LIN {X 0,Y 328.019,Z 1054.025,A -85,B 0,C 180,E1 16291.397,E2 16291.397} C_VEL
LIN {X 0,Y 327.98,Z 1054.756,A -85,B 0,C 180,E1 16287.554,E2 16287.554} C_VEL
LIN {X 0,Y 328.061,Z 1053.985,A -85,B 0,C 180,E1 16283.525,E2 16283.525} C_VEL
LIN {X 0,Y 328.284,Z 1052.234,A -85,B 0,C 180,E1 16280.002,E2 16280.002} C_VEL
LIN {X 0,Y 329.029,Z 1048.812,A -85,B 0,C 180,E1 16275.794,E2 16275.794} C_VEL
LIN {X 0,Y 330.509,Z 1043.751,A -85,B 0,C 180,E1 16271.661,E2 16271.661} C_VEL
LIN {X 0,Y 332.865,Z 1037.506,A -85,B 0,C 180,E1 16267.699,E2 16267.699} C_VEL
LIN {X 0,Y 336.502,Z 1029.05,A -85,B 0,C 180,E1 16263.531,E2 16263.531} C_VEL
LIN {X 0,Y 340.822,Z 1020.018,A -85,B 0,C 180,E1 16259.889,E2 16259.889} C_VEL
LIN {X 0,Y 346.797,Z 1008.189,A -85,B 0,C 180,E1 16255.99,E2 16255.99} C_VEL
LIN {X 0,Y 352.877,Z 996.469,A -85,B 0,C 180,E1 16252.772,E2 16252.772} C_VEL
LIN {X 0,Y 360.668,Z 981.476,A -85,B 0,C 180,E1 16249.345,E2 16249.345} C_VEL
LIN {X 0,Y 367.6,Z 967.844,A -85,B 0,C 180,E1 16246.729,E2 16246.729} C_VEL
LIN {X 0,Y 376.145,Z 950.498,A -85,B 0,C 180,E1 16243.914,E2 16243.914} C_VEL
LIN {X 0,Y 383.701,Z 934.237,A -85,B 0,C 180,E1 16241.704,E2 16241.704} C_VEL
LIN {X 0,Y 392.054,Z 915.275,A -85,B 0,C 180,E1 16239.512,E2 16239.512} C_VEL
LIN {X 0,Y 397.893,Z 900.897,A -85,B 0,C 180,E1 16238.1,E2 16238.1} C_VEL
LIN {X 0,Y 399.57,Z 894.838,A -85,B 0,C 180,E1 16237.443,E2 16237.443} C_VEL
LIN {X 0,Y 401.539,Z 880.043,A -85,B 0,C 180,E1 16235.512,E2 16235.512} C_VEL
LIN {X 0,Y 403.175,Z 873.668,A -85,B 0,C 180,E1 16234.932,E2 16234.932} C_VEL
LIN {X 0,Y 409.897,Z 853.186,A -85,B 0,C 180,E1 16233.587,E2 16233.587} C_VEL
LIN {X 0,Y 416.193,Z 831.541,A -85,B 0,C 180,E1 16232.395,E2 16232.395} C_VEL
LIN {X 0,Y 421.864,Z 808.1,A -85,B 0,C 180,E1 16231.367,E2 16231.367} C_VEL
LIN {X 0,Y 426.386,Z 785.736,A -85,B 0,C 180,E1 16230.586,E2 16230.586} C_VEL
LIN {X 0,Y 430.208,Z 760.734,A -85,B 0,C 180,E1 16229.93,E2 16229.93} C_VEL
LIN {X 0,Y 432.597,Z 738.268,A -85,B 0,C 180,E1 16229.491,E2 16229.491} C_VEL
LIN {X 0,Y 447.979,Z 526.259,A -85,B 0,C 180,E1 16226.067,E2 16226.067} C_VEL
LIN {X 0,Y 439.532,Z 512.486,A -85,B 0,C 180,E1 16223.283,E2 16223.283} C_VEL
LIN {X 0,Y 431.504,Z 500.147,A -85,B 0,C 180,E1 16220.234,E2 16220.234} C_VEL
LIN {X 0,Y 424.951,Z 490.677,A -85,B 0,C 180,E1 16217.317,E2 16217.317} C_VEL
LIN {X 0,Y 420.889,Z 485.14,A -85,B 0,C 180,E1 16215.219,E2 16215.219} C_VEL
LIN {X 0,Y 417.649,Z 480.579,A -85,B 0,C 180,E1 16213.287,E2 16213.287} C_VEL
LIN {X 0,Y 414.017,Z 475.592,A -85,B 0,C 180,E1 16210.717,E2 16210.717} C_VEL
LIN {X 0,Y 410.905,Z 471.414,A -85,B 0,C 180,E1 16207.902,E2 16207.902} C_VEL
LIN {X 0,Y 410.246,Z 470.248,A -85,B 0,C 180,E1 16207.141,E2 16207.141} C_VEL
LIN {X 0,Y 406.911,Z 465.074,A -85,B 0,C 180,E1 16199.437,E2 16199.437} C_VEL
LIN {X 0,Y 406.969,Z 465.799,A -85,B 0,C 180,E1 16197.606,E2 16197.606} C_VEL
LIN {X 0,Y 410.641,Z 470.746,A -85,B 0,C 180,E1 16190.752,E2 16190.752} C_VEL
LIN {X 0,Y 413.009,Z 474.635,A -85,B 0,C 180,E1 16188.408,E2 16188.408} C_VEL
LIN {X 0,Y 414.68,Z 476.395,A -85,B 0,C 180,E1 16187.112,E2 16187.112} C_VEL
LIN {X 0,Y 418.024,Z 480.996,A -85,B 0,C 180,E1 16184.816,E2 16184.816} C_VEL
LIN {X 0,Y 422.672,Z 487.53,A -85,B 0,C 180,E1 16182.16,E2 16182.16} C_VEL
LIN {X 0,Y 426.717,Z 493.371,A -85,B 0,C 180,E1 16180.173,E2 16180.173} C_VEL
LIN {X 0,Y 433.716,Z 505.116,A -85,B 0,C 180,E1 16177.141,E2 16177.141} C_VEL
LIN {X 0,Y 441.286,Z 518.517,A -85,B 0,C 180,E1 16174.32,E2 16174.32} C_VEL
LIN {X 0,Y 447.828,Z 531.14,A -85,B 0,C 180,E1 16172.136,E2 16172.136} C_VEL
LIN {X 0,Y 431.317,Z 757.329,A -85,B 0,C 180,E1 16168.476,E2 16168.476} C_VEL
LIN {X 0,Y 427.838,Z 784.421,A -85,B 0,C 180,E1 16167.9,E2 16167.9} C_VEL
LIN {X 0,Y 423.888,Z 806.262,A -85,B 0,C 180,E1 16167.286,E2 16167.286} C_VEL
LIN {X 0,Y 418.06,Z 831.955,A -85,B 0,C 180,E1 16166.338,E2 16166.338} C_VEL
LIN {X 0,Y 412.513,Z 852.441,A -85,B 0,C 180,E1 16165.378,E2 16165.378} C_VEL
LIN {X 0,Y 405.328,Z 875.569,A -85,B 0,C 180,E1 16164.047,E2 16164.047} C_VEL
LIN {X 0,Y 398.484,Z 894.862,A -85,B 0,C 180,E1 16162.696,E2 16162.696} C_VEL
LIN {X 0,Y 390.831,Z 914.648,A -85,B 0,C 180,E1 16161.055,E2 16161.055} C_VEL
LIN {X 0,Y 382.147,Z 934.931,A -85,B 0,C 180,E1 16159.013,E2 16159.013} C_VEL
LIN {X 0,Y 374.49,Z 951.703,A -85,B 0,C 180,E1 16157.019,E2 16157.019} C_VEL
LIN {X 0,Y 365.624,Z 969.96,A -85,B 0,C 180,E1 16154.435,E2 16154.435} C_VEL
LIN {X 0,Y 357.949,Z 985.105,A -85,B 0,C 180,E1 16151.884,E2 16151.884} C_VEL
LIN {X 0,Y 349.451,Z 1001.499,A -85,B 0,C 180,E1 16148.592,E2 16148.592} C_VEL
LIN {X 0,Y 342.714,Z 1014.35,A -85,B 0,C 180,E1 16145.492,E2 16145.492} C_VEL
LIN {X 0,Y 336.074,Z 1027.324,A -85,B 0,C 180,E1 16141.777,E2 16141.777} C_VEL
LIN {X 0,Y 330.792,Z 1038.04,A -85,B 0,C 180,E1 16138.038,E2 16138.038} C_VEL
LIN {X 0,Y 326.517,Z 1047.639,A -85,B 0,C 180,E1 16134.034,E2 16134.034} C_VEL
LIN {X 0,Y 323.393,Z 1055.523,A -85,B 0,C 180,E1 16129.883,E2 16129.883} C_VEL
LIN {X 0,Y 321.47,Z 1061.654,A -85,B 0,C 180,E1 16125.885,E2 16125.885} C_VEL
LIN {X 0,Y 320.346,Z 1066.696,A -85,B 0,C 180,E1 16121.453,E2 16121.453} C_VEL
LIN {X 0,Y 319.995,Z 1069.639,A -85,B 0,C 180,E1 16117.722,E2 16117.722} C_VEL
LIN {X 0,Y 319.957,Z 1071.386,A -85,B 0,C 180,E1 16114.122,E2 16114.122} C_VEL
LIN {X 0,Y 319.988,Z 1072.022,A -85,B 0,C 180,E1 16110.179,E2 16110.179} C_VEL
LIN {X 0,Y 319.968,Z 1071.269,A -85,B 0,C 180,E1 16106.417,E2 16106.417} C_VEL
LIN {X 0,Y 319.984,Z 1069.557,A -85,B 0,C 180,E1 16103,E2 16103} C_VEL
LIN {X 0,Y 320.217,Z 1066.668,A -85,B 0,C 180,E1 16099.384,E2 16099.384} C_VEL
LIN {X 0,Y 321.182,Z 1061.399,A -85,B 0,C 180,E1 16094.841,E2 16094.841} C_VEL
LIN {X 0,Y 322.786,Z 1055.481,A -85,B 0,C 180,E1 16091.019,E2 16091.019} C_VEL
LIN {X 0,Y 325.582,Z 1047.504,A -85,B 0,C 180,E1 16086.853,E2 16086.853} C_VEL
LIN {X 0,Y 329.389,Z 1038.022,A -85,B 0,C 180,E1 16082.913,E2 16082.913} C_VEL
LIN {X 0,Y 334.287,Z 1027.212,A -85,B 0,C 180,E1 16079.144,E2 16079.144} C_VEL
LIN {X 0,Y 340.353,Z 1014.354,A -85,B 0,C 180,E1 16075.459,E2 16075.459} C_VEL
LIN {X 0,Y 346.711,Z 1001.36,A -85,B 0,C 180,E1 16072.31,E2 16072.31} C_VEL
LIN {X 0,Y 354.366,Z 985.586,A -85,B 0,C 180,E1 16069.109,E2 16069.109} C_VEL
LIN {X 0,Y 361.656,Z 970.313,A -85,B 0,C 180,E1 16066.495,E2 16066.495} C_VEL
LIN {X 0,Y 370.629,Z 950.761,A -85,B 0,C 180,E1 16063.696,E2 16063.696} C_VEL
LIN {X 0,Y 377.757,Z 934.31,A -85,B 0,C 180,E1 16061.718,E2 16061.718} C_VEL
LIN {X 0,Y 386.147,Z 913.615,A -85,B 0,C 180,E1 16059.615,E2 16059.615} C_VEL
LIN {X 0,Y 392.979,Z 895.121,A -85,B 0,C 180,E1 16058.049,E2 16058.049} C_VEL
LIN {X 0,Y 400.135,Z 874.089,A -85,B 0,C 180,E1 16056.545,E2 16056.545} C_VEL
LIN {X 0,Y 406.584,Z 852.194,A -85,B 0,C 180,E1 16055.267,E2 16055.267} C_VEL
LIN {X 0,Y 411.987,Z 831.39,A -85,B 0,C 180,E1 16054.268,E2 16054.268} C_VEL
LIN {X 0,Y 417.472,Z 806.131,A -85,B 0,C 180,E1 16053.315,E2 16053.315} C_VEL
LIN {X 0,Y 421.276,Z 784.291,A -85,B 0,C 180,E1 16052.684,E2 16052.684} C_VEL
LIN {X 0,Y 424.587,Z 757.418,A -85,B 0,C 180,E1 16052.1,E2 16052.1} C_VEL
LIN {X 0,Y 440.37,Z 531.132,A -85,B 0,C 180,E1 16048.393,E2 16048.393} C_VEL
LIN {X 0,Y 440.634,Z 526.173,A -85,B 0,C 180,E1 16048.293,E2 16048.293} C_VEL
LIN {X 0,Y 432.575,Z 510.753,A -85,B 0,C 180,E1 16045.794,E2 16045.794} C_VEL
LIN {X 0,Y 424.816,Z 497.033,A -85,B 0,C 180,E1 16043.109,E2 16043.109} C_VEL
LIN {X 0,Y 418.086,Z 485.932,A -85,B 0,C 180,E1 16040.473,E2 16040.473} C_VEL
LIN {X 0,Y 412.337,Z 477.708,A -85,B 0,C 180,E1 16037.937,E2 16037.937} C_VEL
LIN {X 0,Y 407.928,Z 471.833,A -85,B 0,C 180,E1 16035.715,E2 16035.715} C_VEL
LIN {X 0,Y 404.622,Z 467.31,A -85,B 0,C 180,E1 16033.796,E2 16033.796} C_VEL
LIN {X 0,Y 401.321,Z 462.864,A -85,B 0,C 180,E1 16031.57,E2 16031.57} C_VEL
LIN {X 0,Y 397.458,Z 458.072,A -85,B 0,C 180,E1 16028.317,E2 16028.317} C_VEL
LIN {X 0,Y 396.63,Z 456.484,A -85,B 0,C 180,E1 16027.387,E2 16027.387} C_VEL
LIN {X 0,Y 393.119,Z 452.323,A -85,B 0,C 180,E1 16021.457,E2 16021.457} C_VEL
LIN {X 0,Y 392.894,Z 450.705,A -85,B 0,C 180,E1 16018.833,E2 16018.833} C_VEL
LIN {X 0,Y 393.131,Z 452.387,A -85,B 0,C 180,E1 16016.062,E2 16016.062} C_VEL
LIN {X 0,Y 396.418,Z 456.356,A -85,B 0,C 180,E1 16010.417,E2 16010.417} C_VEL
LIN {X 0,Y 397.008,Z 457.086,A -85,B 0,C 180,E1 16009.772,E2 16009.772} C_VEL
LIN {X 0,Y 399.817,Z 461.29,A -85,B 0,C 180,E1 16007.139,E2 16007.139} C_VEL
LIN {X 0,Y 401.324,Z 462.818,A -85,B 0,C 180,E1 16006.015,E2 16006.015} C_VEL
LIN {X 0,Y 404.74,Z 467.435,A -85,B 0,C 180,E1 16003.716,E2 16003.716} C_VEL
LIN {X 0,Y 409.748,Z 474.244,A -85,B 0,C 180,E1 16000.913,E2 16000.913} C_VEL
LIN {X 0,Y 413.929,Z 480.014,A -85,B 0,C 180,E1 15998.904,E2 15998.904} C_VEL
LIN {X 0,Y 419.585,Z 487.91,A -85,B 0,C 180,E1 15996.511,E2 15996.511} C_VEL
LIN {X 0,Y 428.149,Z 500.756,A -85,B 0,C 180,E1 15993.359,E2 15993.359} C_VEL
LIN {X 0,Y 436.584,Z 514.241,A -85,B 0,C 180,E1 15990.652,E2 15990.652} C_VEL
LIN {X 0,Y 440.881,Z 521.726,A -85,B 0,C 180,E1 15989.377,E2 15989.377} C_VEL
LIN {X 0,Y 425.191,Z 745.395,A -85,B 0,C 180,E1 15985.721,E2 15985.721} C_VEL
LIN {X 0,Y 421.987,Z 771.99,A -85,B 0,C 180,E1 15985.121,E2 15985.121} C_VEL
LIN {X 0,Y 418.53,Z 792.778,A -85,B 0,C 180,E1 15984.488,E2 15984.488} C_VEL
LIN {X 0,Y 413.739,Z 816.139,A -85,B 0,C 180,E1 15983.588,E2 15983.588} C_VEL
LIN {X 0,Y 408.538,Z 836.869,A -85,B 0,C 180,E1 15982.581,E2 15982.581} C_VEL
LIN {X 0,Y 402.594,Z 857.714,A -85,B 0,C 180,E1 15981.361,E2 15981.361} C_VEL
LIN {X 0,Y 395.356,Z 879.706,A -85,B 0,C 180,E1 15979.799,E2 15979.799} C_VEL
LIN {X 0,Y 388.487,Z 898.569,A -85,B 0,C 180,E1 15978.193,E2 15978.193} C_VEL
LIN {X 0,Y 379.969,Z 919.801,A -85,B 0,C 180,E1 15976.031,E2 15976.031} C_VEL
LIN {X 0,Y 372.729,Z 936.462,A -85,B 0,C 180,E1 15974.011,E2 15974.011} C_VEL
LIN {X 0,Y 364.37,Z 954.654,A -85,B 0,C 180,E1 15971.402,E2 15971.402} C_VEL
LIN {X 0,Y 357.091,Z 969.614,A -85,B 0,C 180,E1 15968.845,E2 15968.845} C_VEL
LIN {X 0,Y 349.753,Z 984.458,A -85,B 0,C 180,E1 15965.878,E2 15965.878} C_VEL
LIN {X 0,Y 342.642,Z 998.396,A -85,B 0,C 180,E1 15962.504,E2 15962.504} C_VEL
LIN {X 0,Y 336.519,Z 1010.737,A -85,B 0,C 180,E1 15958.968,E2 15958.968} C_VEL
LIN {X 0,Y 331.261,Z 1021.518,A -85,B 0,C 180,E1 15955.189,E2 15955.189} C_VEL
LIN {X 0,Y 327.31,Z 1030.305,A -85,B 0,C 180,E1 15951.505,E2 15951.505} C_VEL
LIN {X 0,Y 324.001,Z 1038.513,A -85,B 0,C 180,E1 15947.233,E2 15947.233} C_VEL
LIN {X 0,Y 322.06,Z 1044.254,A -85,B 0,C 180,E1 15943.465,E2 15943.465} C_VEL
LIN {X 0,Y 320.745,Z 1049.314,A -85,B 0,C 180,E1 15939.148,E2 15939.148} C_VEL
LIN {X 0,Y 320.194,Z 1052.426,A -85,B 0,C 180,E1 15935.196,E2 15935.196} C_VEL
LIN {X 0,Y 320.025,Z 1054.183,A -85,B 0,C 180,E1 15931.611,E2 15931.611} C_VEL
LIN {X 0,Y 319.981,Z 1054.932,A -85,B 0,C 180,E1 15927.851,E2 15927.851} C_VEL
LIN {X 0,Y 320.057,Z 1054.321,A -85,B 0,C 180,E1 15923.723,E2 15923.723} C_VEL
LIN {X 0,Y 320.28,Z 1052.653,A -85,B 0,C 180,E1 15920.113,E2 15920.113} C_VEL
LIN {X 0,Y 320.904,Z 1049.772,A -85,B 0,C 180,E1 15916.302,E2 15916.302} C_VEL
LIN {X 0,Y 322.467,Z 1044.677,A -85,B 0,C 180,E1 15911.749,E2 15911.749} C_VEL
LIN {X 0,Y 324.668,Z 1038.967,A -85,B 0,C 180,E1 15907.931,E2 15907.931} C_VEL
LIN {X 0,Y 328.361,Z 1030.807,A -85,B 0,C 180,E1 15903.603,E2 15903.603} C_VEL
LIN {X 0,Y 332.715,Z 1021.981,A -85,B 0,C 180,E1 15899.876,E2 15899.876} C_VEL
LIN {X 0,Y 338.485,Z 1011.156,A -85,B 0,C 180,E1 15896.061,E2 15896.061} C_VEL
LIN {X 0,Y 345.089,Z 998.802,A -85,B 0,C 180,E1 15892.521,E2 15892.521} C_VEL
LIN {X 0,Y 352.564,Z 985.141,A -85,B 0,C 180,E1 15889.221,E2 15889.221} C_VEL
LIN {X 0,Y 360.305,Z 970.456,A -85,B 0,C 180,E1 15886.29,E2 15886.29} C_VEL
LIN {X 0,Y 368.073,Z 955.375,A -85,B 0,C 180,E1 15883.73,E2 15883.73} C_VEL
LIN {X 0,Y 376.988,Z 937.051,A -85,B 0,C 180,E1 15881.127,E2 15881.127} C_VEL
LIN {X 0,Y 384.682,Z 920.217,A -85,B 0,C 180,E1 15879.115,E2 15879.115} C_VEL
LIN {X 0,Y 393.636,Z 898.972,A -85,B 0,C 180,E1 15876.989,E2 15876.989} C_VEL
LIN {X 0,Y 400.704,Z 880.424,A -85,B 0,C 180,E1 15875.44,E2 15875.44} C_VEL
LIN {X 0,Y 403.175,Z 873.668,A -85,B 0,C 180,E1 15874.932,E2 15874.932} C_VEL
LIN {X 0,Y 404.8,Z 867.191,A -85,B 0,C 180,E1 15874.368,E2 15874.368} C_VEL
LIN {X 0,Y 406.692,Z 851.349,A -85,B 0,C 180,E1 15872.637,E2 15872.637} C_VEL
LIN {X 0,Y 408.136,Z 844.614,A -85,B 0,C 180,E1 15872.138,E2 15872.138} C_VEL
LIN {X 0,Y 413.973,Z 823.428,A -85,B 0,C 180,E1 15871.078,E2 15871.078} C_VEL
LIN {X 0,Y 418.898,Z 802.662,A -85,B 0,C 180,E1 15870.223,E2 15870.223} C_VEL
LIN {X 0,Y 423.613,Z 777.831,A -85,B 0,C 180,E1 15869.427,E2 15869.427} C_VEL
LIN {X 0,Y 426.807,Z 755.743,A -85,B 0,C 180,E1 15868.893,E2 15868.893} C_VEL
LIN {X 0,Y 429.76,Z 723.203,A -85,B 0,C 180,E1 15868.317,E2 15868.317} C_VEL
LIN {X 0,Y 444.069,Z 530.795,A -85,B 0,C 180,E1 15865.222,E2 15865.222} C_VEL
LIN {X 0,Y 436.41,Z 518.249,A -85,B 0,C 180,E1 15862.587,E2 15862.587} C_VEL
LIN {X 0,Y 429.334,Z 507.17,A -85,B 0,C 180,E1 15859.799,E2 15859.799} C_VEL
LIN {X 0,Y 423.024,Z 497.889,A -85,B 0,C 180,E1 15856.902,E2 15856.902} C_VEL
LIN {X 0,Y 419.308,Z 492.682,A -85,B 0,C 180,E1 15854.924,E2 15854.924} C_VEL
LIN {X 0,Y 416.245,Z 488.267,A -85,B 0,C 180,E1 15853.05,E2 15853.05} C_VEL
LIN {X 0,Y 412.688,Z 483.313,A -85,B 0,C 180,E1 15850.47,E2 15850.47} C_VEL
LIN {X 0,Y 409.67,Z 479.099,A -85,B 0,C 180,E1 15847.644,E2 15847.644} C_VEL
LIN {X 0,Y 409.147,Z 478.135,A -85,B 0,C 180,E1 15847.019,E2 15847.019} C_VEL
LIN {X 0,Y 405.936,Z 472.985,A -85,B 0,C 180,E1 15839.294,E2 15839.294} C_VEL
LIN {X 0,Y 406.126,Z 474.378,A -85,B 0,C 180,E1 15836.754,E2 15836.754} C_VEL
LIN {X 0,Y 409.473,Z 478.582,A -85,B 0,C 180,E1 15830.938,E2 15830.938} C_VEL
LIN {X 0,Y 411.873,Z 482.526,A -85,B 0,C 180,E1 15828.517,E2 15828.517} C_VEL
LIN {X 0,Y 413.425,Z 484.272,A -85,B 0,C 180,E1 15827.286,E2 15827.286} C_VEL
LIN {X 0,Y 417.461,Z 489.989,A -85,B 0,C 180,E1 15824.51,E2 15824.51} C_VEL
LIN {X 0,Y 421.183,Z 495.284,A -85,B 0,C 180,E1 15822.381,E2 15822.381} C_VEL
LIN {X 0,Y 424.826,Z 500.638,A -85,B 0,C 180,E1 15820.546,E2 15820.546} C_VEL
LIN {X 0,Y 432.308,Z 513.406,A -85,B 0,C 180,E1 15817.242,E2 15817.242} C_VEL
LIN {X 0,Y 440.672,Z 528.855,A -85,B 0,C 180,E1 15814.101,E2 15814.101} C_VEL
LIN {X 0,Y 443.886,Z 535.634,A -85,B 0,C 180,E1 15812.986,E2 15812.986} C_VEL
LIN {X 0,Y 427.242,Z 757.597,A -85,B 0,C 180,E1 15809.395,E2 15809.395} C_VEL
LIN {X 0,Y 423.71,Z 784.37,A -85,B 0,C 180,E1 15808.825,E2 15808.825} C_VEL
LIN {X 0,Y 419.68,Z 806.184,A -85,B 0,C 180,E1 15808.215,E2 15808.215} C_VEL
LIN {X 0,Y 413.842,Z 831.412,A -85,B 0,C 180,E1 15807.292,E2 15807.292} C_VEL
LIN {X 0,Y 408.322,Z 851.396,A -85,B 0,C 180,E1 15806.365,E2 15806.365} C_VEL
LIN {X 0,Y 401.506,Z 873.159,A -85,B 0,C 180,E1 15805.142,E2 15805.142} C_VEL
LIN {X 0,Y 393.932,Z 894.049,A -85,B 0,C 180,E1 15803.696,E2 15803.696} C_VEL
LIN {X 0,Y 386.349,Z 913.156,A -85,B 0,C 180,E1 15802.125,E2 15802.125} C_VEL
LIN {X 0,Y 377.4,Z 933.656,A -85,B 0,C 180,E1 15800.086,E2 15800.086} C_VEL
LIN {X 0,Y 369.476,Z 950.519,A -85,B 0,C 180,E1 15798.092,E2 15798.092} C_VEL
LIN {X 0,Y 359.799,Z 969.863,A -85,B 0,C 180,E1 15795.351,E2 15795.351} C_VEL
LIN {X 0,Y 351.855,Z 984.997,A -85,B 0,C 180,E1 15792.78,E2 15792.78} C_VEL
LIN {X 0,Y 342.877,Z 1001.628,A -85,B 0,C 180,E1 15789.395,E2 15789.395} C_VEL
LIN {X 0,Y 336.005,Z 1014.213,A -85,B 0,C 180,E1 15786.312,E2 15786.312} C_VEL
LIN {X 0,Y 329.057,Z 1027.171,A -85,B 0,C 180,E1 15782.537,E2 15782.537} C_VEL
LIN {X 0,Y 323.621,Z 1037.65,A -85,B 0,C 180,E1 15778.816,E2 15778.816} C_VEL
LIN {X 0,Y 318.968,Z 1047.503,A -85,B 0,C 180,E1 15774.621,E2 15774.621} C_VEL
LIN {X 0,Y 315.623,Z 1055.451,A -85,B 0,C 180,E1 15770.326,E2 15770.326} C_VEL
LIN {X 0,Y 313.538,Z 1061.728,A -85,B 0,C 180,E1 15766.108,E2 15766.108} C_VEL
LIN {X 0,Y 312.37,Z 1066.613,A -85,B 0,C 180,E1 15761.62,E2 15761.62} C_VEL
LIN {X 0,Y 312.001,Z 1069.438,A -85,B 0,C 180,E1 15757.921,E2 15757.921} C_VEL
LIN {X 0,Y 311.959,Z 1071.181,A -85,B 0,C 180,E1 15754.228,E2 15754.228} C_VEL
LIN {X 0,Y 311.991,Z 1071.805,A -85,B 0,C 180,E1 15750.184,E2 15750.184} C_VEL
LIN {X 0,Y 311.968,Z 1071.047,A -85,B 0,C 180,E1 15746.325,E2 15746.325} C_VEL
LIN {X 0,Y 311.998,Z 1069.328,A -85,B 0,C 180,E1 15742.82,E2 15742.82} C_VEL
LIN {X 0,Y 312.25,Z 1066.432,A -85,B 0,C 180,E1 15739.11,E2 15739.11} C_VEL
LIN {X 0,Y 313.297,Z 1061.149,A -85,B 0,C 180,E1 15734.45,E2 15734.45} C_VEL
LIN {X 0,Y 315.039,Z 1055.168,A -85,B 0,C 180,E1 15730.5,E2 15730.5} C_VEL
LIN {X 0,Y 318.158,Z 1046.817,A -85,B 0,C 180,E1 15726.083,E2 15726.083} C_VEL
LIN {X 0,Y 322.247,Z 1037.273,A -85,B 0,C 180,E1 15722.061,E2 15722.061} C_VEL
LIN {X 0,Y 327.593,Z 1026.099,A -85,B 0,C 180,E1 15718.127,E2 15718.127} C_VEL
LIN {X 0,Y 333.87,Z 1013.402,A -85,B 0,C 180,E1 15714.479,E2 15714.479} C_VEL
LIN {X 0,Y 340.927,Z 999.62,A -85,B 0,C 180,E1 15711.125,E2 15711.125} C_VEL
LIN {X 0,Y 348.565,Z 984.395,A -85,B 0,C 180,E1 15708.058,E2 15708.058} C_VEL
LIN {X 0,Y 356.173,Z 969.031,A -85,B 0,C 180,E1 15705.426,E2 15705.426} C_VEL
LIN {X 0,Y 364.98,Z 950.393,A -85,B 0,C 180,E1 15702.76,E2 15702.76} C_VEL
LIN {X 0,Y 372.335,Z 933.928,A -85,B 0,C 180,E1 15700.773,E2 15700.773} C_VEL
LIN {X 0,Y 381.032,Z 913.033,A -85,B 0,C 180,E1 15698.649,E2 15698.649} C_VEL
LIN {X 0,Y 388.104,Z 894.392,A -85,B 0,C 180,E1 15697.076,E2 15697.076} C_VEL
LIN {X 0,Y 395.647,Z 872.679,A -85,B 0,C 180,E1 15695.535,E2 15695.535} C_VEL
LIN {X 0,Y 402.205,Z 850.772,A -85,B 0,C 180,E1 15694.275,E2 15694.275} C_VEL
LIN {X 0,Y 408.035,Z 828.711,A -85,B 0,C 180,E1 15693.235,E2 15693.235} C_VEL
LIN {X 0,Y 413.218,Z 804.801,A -85,B 0,C 180,E1 15692.358,E2 15692.358} C_VEL
LIN {X 0,Y 417.156,Z 782.419,A -85,B 0,C 180,E1 15691.722,E2 15691.722} C_VEL
LIN {X 0,Y 420.314,Z 756.611,A -85,B 0,C 180,E1 15691.171,E2 15691.171} C_VEL
LIN {X 0,Y 436.53,Z 530.272,A -85,B 0,C 180,E1 15687.462,E2 15687.462} C_VEL
LIN {X 0,Y 428.636,Z 515.087,A -85,B 0,C 180,E1 15684.901,E2 15684.901} C_VEL
LIN {X 0,Y 421.73,Z 502.799,A -85,B 0,C 180,E1 15682.404,E2 15682.404} C_VEL
LIN {X 0,Y 415.985,Z 493.07,A -85,B 0,C 180,E1 15680.067,E2 15680.067} C_VEL
LIN {X 0,Y 410.36,Z 484.919,A -85,B 0,C 180,E1 15677.513,E2 15677.513} C_VEL
LIN {X 0,Y 406.316,Z 479.373,A -85,B 0,C 180,E1 15675.413,E2 15675.413} C_VEL
LIN {X 0,Y 403.078,Z 474.887,A -85,B 0,C 180,E1 15673.484,E2 15673.484} C_VEL
LIN {X 0,Y 399.782,Z 470.229,A -85,B 0,C 180,E1 15671.177,E2 15671.177} C_VEL
LIN {X 0,Y 396.394,Z 466.147,A -85,B 0,C 180,E1 15668.267,E2 15668.267} C_VEL
LIN {X 0,Y 395.52,Z 464.374,A -85,B 0,C 180,E1 15667.262,E2 15667.262} C_VEL
LIN {X 0,Y 392.107,Z 460.199,A -85,B 0,C 180,E1 15661.315,E2 15661.315} C_VEL
LIN {X 0,Y 391.923,Z 458.619,A -85,B 0,C 180,E1 15658.684,E2 15658.684} C_VEL
LIN {X 0,Y 395.453,Z 464.321,A -85,B 0,C 180,E1 15650.394,E2 15650.394} C_VEL
LIN {X 0,Y 398.852,Z 469.35,A -85,B 0,C 180,E1 15647.108,E2 15647.108} C_VEL
LIN {X 0,Y 400.055,Z 470.705,A -85,B 0,C 180,E1 15646.191,E2 15646.191} C_VEL
LIN {X 0,Y 404.204,Z 476.438,A -85,B 0,C 180,E1 15643.398,E2 15643.398} C_VEL
LIN {X 0,Y 408.109,Z 481.813,A -85,B 0,C 180,E1 15641.205,E2 15641.205} C_VEL
LIN {X 0,Y 412.144,Z 487.49,A -85,B 0,C 180,E1 15639.218,E2 15639.218} C_VEL
LIN {X 0,Y 417.683,Z 495.416,A -85,B 0,C 180,E1 15636.818,E2 15636.818} C_VEL
LIN {X 0,Y 425.779,Z 507.797,A -85,B 0,C 180,E1 15633.763,E2 15633.763} C_VEL
LIN {X 0,Y 433.973,Z 521.148,A -85,B 0,C 180,E1 15631.063,E2 15631.063} C_VEL
LIN {X 0,Y 436.683,Z 526.126,A -85,B 0,C 180,E1 15630.223,E2 15630.223} C_VEL
LIN {X 0,Y 420.829,Z 746.012,A -85,B 0,C 180,E1 15626.625,E2 15626.625} C_VEL
LIN {X 0,Y 417.528,Z 772.58,A -85,B 0,C 180,E1 15626.024,E2 15626.024} C_VEL
LIN {X 0,Y 413.994,Z 793.305,A -85,B 0,C 180,E1 15625.393,E2 15625.393} C_VEL
LIN {X 0,Y 408.88,Z 817.43,A -85,B 0,C 180,E1 15624.456,E2 15624.456} C_VEL
LIN {X 0,Y 403.422,Z 838.547,A -85,B 0,C 180,E1 15623.421,E2 15623.421} C_VEL
LIN {X 0,Y 396.748,Z 861.148,A -85,B 0,C 180,E1 15622.076,E2 15622.076} C_VEL
LIN {X 0,Y 389.639,Z 881.774,A -85,B 0,C 180,E1 15620.572,E2 15620.572} C_VEL
LIN {X 0,Y 382.034,Z 901.996,A -85,B 0,C 180,E1 15618.816,E2 15618.816} C_VEL
LIN {X 0,Y 373.957,Z 921.227,A -85,B 0,C 180,E1 15616.804,E2 15616.804} C_VEL
LIN {X 0,Y 366.455,Z 937.947,A -85,B 0,C 180,E1 15614.746,E2 15614.746} C_VEL
LIN {X 0,Y 357.859,Z 955.928,A -85,B 0,C 180,E1 15612.112,E2 15612.112} C_VEL
LIN {X 0,Y 350.795,Z 969.964,A -85,B 0,C 180,E1 15609.678,E2 15609.678} C_VEL
LIN {X 0,Y 343.188,Z 984.792,A -85,B 0,C 180,E1 15606.675,E2 15606.675} C_VEL
LIN {X 0,Y 336.074,Z 998.178,A -85,B 0,C 180,E1 15603.395,E2 15603.395} C_VEL
LIN {X 0,Y 329.965,Z 1009.92,A -85,B 0,C 180,E1 15600,E2 15600} C_VEL
LIN {X 0,Y 324.125,Z 1021.359,A -85,B 0,C 180,E1 15595.98,E2 15595.98} C_VEL
LIN {X 0,Y 319.921,Z 1030.19,A -85,B 0,C 180,E1 15592.221,E2 15592.221} C_VEL
LIN {X 0,Y 316.256,Z 1038.778,A -85,B 0,C 180,E1 15587.669,E2 15587.669} C_VEL
LIN {X 0,Y 314.196,Z 1044.51,A -85,B 0,C 180,E1 15583.808,E2 15583.808} C_VEL
LIN {X 0,Y 312.799,Z 1049.554,A -85,B 0,C 180,E1 15579.383,E2 15579.383} C_VEL
LIN {X 0,Y 312.21,Z 1052.658,A -85,B 0,C 180,E1 15575.329,E2 15575.329} C_VEL
LIN {X 0,Y 312.029,Z 1054.407,A -85,B 0,C 180,E1 15571.653,E2 15571.653} C_VEL
LIN {X 0,Y 311.984,Z 1055.15,A -85,B 0,C 180,E1 15567.796,E2 15567.796} C_VEL
LIN {X 0,Y 312.068,Z 1054.525,A -85,B 0,C 180,E1 15563.561,E2 15563.561} C_VEL
LIN {X 0,Y 312.31,Z 1052.851,A -85,B 0,C 180,E1 15559.858,E2 15559.858} C_VEL
LIN {X 0,Y 312.996,Z 1049.964,A -85,B 0,C 180,E1 15555.949,E2 15555.949} C_VEL
LIN {X 0,Y 314.708,Z 1044.785,A -85,B 0,C 180,E1 15551.229,E2 15551.229} C_VEL
LIN {X 0,Y 317.043,Z 1039.138,A -85,B 0,C 180,E1 15547.371,E2 15547.371} C_VEL
LIN {X 0,Y 320.972,Z 1030.962,A -85,B 0,C 180,E1 15542.947,E2 15542.947} C_VEL
LIN {X 0,Y 325.565,Z 1022.129,A -85,B 0,C 180,E1 15539.143,E2 15539.143} C_VEL
LIN {X 0,Y 331.629,Z 1011.288,A -85,B 0,C 180,E1 15535.26,E2 15535.26} C_VEL
LIN {X 0,Y 338.541,Z 998.922,A -85,B 0,C 180,E1 15531.666,E2 15531.666} C_VEL
LIN {X 0,Y 346.21,Z 985.46,A -85,B 0,C 180,E1 15528.374,E2 15528.374} C_VEL
LIN {X 0,Y 354.624,Z 970.07,A -85,B 0,C 180,E1 15525.279,E2 15525.279} C_VEL
LIN {X 0,Y 363.408,Z 953.602,A -85,B 0,C 180,E1 15522.491,E2 15522.491} C_VEL
LIN {X 0,Y 372.16,Z 935.987,A -85,B 0,C 180,E1 15520.029,E2 15520.029} C_VEL
LIN {X 0,Y 380.693,Z 917.814,A -85,B 0,C 180,E1 15517.883,E2 15517.883} C_VEL
LIN {X 0,Y 389.097,Z 898.152,A -85,B 0,C 180,E1 15515.955,E2 15515.955} C_VEL
LIN {X 0,Y 396.341,Z 879.576,A -85,B 0,C 180,E1 15514.416,E2 15514.416} C_VEL
LIN {X 0,Y 404.502,Z 856.112,A -85,B 0,C 180,E1 15512.813,E2 15512.813} C_VEL
LIN {X 0,Y 408.136,Z 844.614,A -85,B 0,C 180,E1 15512.138,E2 15512.138} C_VEL
LIN {X 0,Y 409.545,Z 837.786,A -85,B 0,C 180,E1 15511.656,E2 15511.656} C_VEL
LIN {X 0,Y 411.055,Z 821.016,A -85,B 0,C 180,E1 15510.118,E2 15510.118} C_VEL
LIN {X 0,Y 412.236,Z 813.969,A -85,B 0,C 180,E1 15509.702,E2 15509.702} C_VEL
LIN {X 0,Y 417.168,Z 791.338,A -85,B 0,C 180,E1 15508.884,E2 15508.884} C_VEL
LIN {X 0,Y 421.227,Z 768.374,A -85,B 0,C 180,E1 15508.233,E2 15508.233} C_VEL
LIN {X 0,Y 424.198,Z 743.776,A -85,B 0,C 180,E1 15507.722,E2 15507.722} C_VEL
LIN {X 0,Y 440.243,Z 535.419,A -85,B 0,C 180,E1 15504.361,E2 15504.361} C_VEL
LIN {X 0,Y 432.705,Z 522.887,A -85,B 0,C 180,E1 15501.628,E2 15501.628} C_VEL
LIN {X 0,Y 425.772,Z 512.089,A -85,B 0,C 180,E1 15498.732,E2 15498.732} C_VEL
LIN {X 0,Y 420.737,Z 504.576,A -85,B 0,C 180,E1 15496.286,E2 15496.286} C_VEL
LIN {X 0,Y 417.623,Z 500.075,A -85,B 0,C 180,E1 15494.56,E2 15494.56} C_VEL
LIN {X 0,Y 414.64,Z 495.722,A -85,B 0,C 180,E1 15492.676,E2 15492.676} C_VEL
LIN {X 0,Y 411.54,Z 491.193,A -85,B 0,C 180,E1 15490.358,E2 15490.358} C_VEL
LIN {X 0,Y 408.5,Z 486.912,A -85,B 0,C 180,E1 15487.454,E2 15487.454} C_VEL
LIN {X 0,Y 407.925,Z 485.949,A -85,B 0,C 180,E1 15486.757,E2 15486.757} C_VEL
LIN {X 0,Y 404.96,Z 480.934,A -85,B 0,C 180,E1 15479.293,E2 15479.293} C_VEL
LIN {X 0,Y 405.174,Z 482.493,A -85,B 0,C 180,E1 15476.605,E2 15476.605} C_VEL
LIN {X 0,Y 408.31,Z 486.414,A -85,B 0,C 180,E1 15471.125,E2 15471.125} C_VEL
LIN {X 0,Y 410.739,Z 490.415,A -85,B 0,C 180,E1 15468.628,E2 15468.628} C_VEL
LIN {X 0,Y 412.175,Z 492.139,A -85,B 0,C 180,E1 15467.46,E2 15467.46} C_VEL
LIN {X 0,Y 416.043,Z 497.712,A -85,B 0,C 180,E1 15464.742,E2 15464.742} C_VEL
LIN {X 0,Y 419.58,Z 502.842,A -85,B 0,C 180,E1 15462.669,E2 15462.669} C_VEL
LIN {X 0,Y 423.084,Z 508.142,A -85,B 0,C 180,E1 15460.858,E2 15460.858} C_VEL
LIN {X 0,Y 430.274,Z 520.703,A -85,B 0,C 180,E1 15457.597,E2 15457.597} C_VEL
LIN {X 0,Y 438.135,Z 535.607,A -85,B 0,C 180,E1 15454.557,E2 15454.557} C_VEL
LIN {X 0,Y 440.062,Z 539.907,A -85,B 0,C 180,E1 15453.855,E2 15453.855} C_VEL
LIN {X 0,Y 423.319,Z 757.439,A -85,B 0,C 180,E1 15450.339,E2 15450.339} C_VEL
LIN {X 0,Y 419.717,Z 784.19,A -85,B 0,C 180,E1 15449.772,E2 15449.772} C_VEL
LIN {X 0,Y 415.608,Z 805.997,A -85,B 0,C 180,E1 15449.167,E2 15449.167} C_VEL
LIN {X 0,Y 409.689,Z 831.066,A -85,B 0,C 180,E1 15448.257,E2 15448.257} C_VEL
LIN {X 0,Y 403.918,Z 851.482,A -85,B 0,C 180,E1 15447.316,E2 15447.316} C_VEL
LIN {X 0,Y 396.612,Z 874.086,A -85,B 0,C 180,E1 15446.041,E2 15446.041} C_VEL
LIN {X 0,Y 389.187,Z 894.048,A -85,B 0,C 180,E1 15444.658,E2 15444.658} C_VEL
LIN {X 0,Y 381.105,Z 913.869,A -85,B 0,C 180,E1 15443.026,E2 15443.026} C_VEL
LIN {X 0,Y 372.228,Z 933.564,A -85,B 0,C 180,E1 15441.054,E2 15441.054} C_VEL
LIN {X 0,Y 364.051,Z 950.448,A -85,B 0,C 180,E1 15439.052,E2 15439.052} C_VEL
LIN {X 0,Y 354.07,Z 969.767,A -85,B 0,C 180,E1 15436.298,E2 15436.298} C_VEL
LIN {X 0,Y 345.849,Z 984.889,A -85,B 0,C 180,E1 15433.708,E2 15433.708} C_VEL
LIN {X 0,Y 336.675,Z 1001.243,A -85,B 0,C 180,E1 15430.349,E2 15430.349} C_VEL
LIN {X 0,Y 329.367,Z 1014.076,A -85,B 0,C 180,E1 15427.166,E2 15427.166} C_VEL
LIN {X 0,Y 322.102,Z 1027.018,A -85,B 0,C 180,E1 15423.33,E2 15423.33} C_VEL
LIN {X 0,Y 316.389,Z 1037.489,A -85,B 0,C 180,E1 15419.539,E2 15419.539} C_VEL
LIN {X 0,Y 311.489,Z 1047.292,A -85,B 0,C 180,E1 15415.273,E2 15415.273} C_VEL
LIN {X 0,Y 307.959,Z 1055.162,A -85,B 0,C 180,E1 15410.925,E2 15410.925} C_VEL
LIN {X 0,Y 305.682,Z 1061.542,A -85,B 0,C 180,E1 15406.534,E2 15406.534} C_VEL
LIN {X 0,Y 304.419,Z 1066.404,A -85,B 0,C 180,E1 15401.942,E2 15401.942} C_VEL
LIN {X 0,Y 304.013,Z 1069.246,A -85,B 0,C 180,E1 15398.115,E2 15398.115} C_VEL
LIN {X 0,Y 303.96,Z 1071.045,A -85,B 0,C 180,E1 15394.15,E2 15394.15} C_VEL
LIN {X 0,Y 304.002,Z 1071.567,A -85,B 0,C 180,E1 15390,E2 15390} C_VEL
LIN {X 0,Y 303.97,Z 1070.824,A -85,B 0,C 180,E1 15386.228,E2 15386.228} C_VEL
LIN {X 0,Y 304.002,Z 1069.099,A -85,B 0,C 180,E1 15382.63,E2 15382.63} C_VEL
LIN {X 0,Y 304.317,Z 1066.031,A -85,B 0,C 180,E1 15378.63,E2 15378.63} C_VEL
LIN {X 0,Y 305.49,Z 1060.637,A -85,B 0,C 180,E1 15373.847,E2 15373.847} C_VEL
LIN {X 0,Y 307.385,Z 1054.653,A -85,B 0,C 180,E1 15369.83,E2 15369.83} C_VEL
LIN {X 0,Y 310.78,Z 1046.13,A -85,B 0,C 180,E1 15365.276,E2 15365.276} C_VEL
LIN {X 0,Y 314.948,Z 1036.991,A -85,B 0,C 180,E1 15361.354,E2 15361.354} C_VEL
LIN {X 0,Y 320.569,Z 1025.802,A -85,B 0,C 180,E1 15357.343,E2 15357.343} C_VEL
LIN {X 0,Y 327.144,Z 1013.096,A -85,B 0,C 180,E1 15353.634,E2 15353.634} C_VEL
LIN {X 0,Y 334.671,Z 998.993,A -85,B 0,C 180,E1 15350.16,E2 15350.16} C_VEL
LIN {X 0,Y 342.892,Z 983.203,A -85,B 0,C 180,E1 15346.972,E2 15346.972} C_VEL
LIN {X 0,Y 351.564,Z 966.327,A -85,B 0,C 180,E1 15344.099,E2 15344.099} C_VEL
LIN {X 0,Y 359.956,Z 948.899,A -85,B 0,C 180,E1 15341.649,E2 15341.649} C_VEL
LIN {X 0,Y 367.87,Z 931.67,A -85,B 0,C 180,E1 15339.59,E2 15339.59} C_VEL
LIN {X 0,Y 376.774,Z 910.555,A -85,B 0,C 180,E1 15337.487,E2 15337.487} C_VEL
LIN {X 0,Y 383.859,Z 892.297,A -85,B 0,C 180,E1 15335.972,E2 15335.972} C_VEL
LIN {X 0,Y 391.912,Z 869.15,A -85,B 0,C 180,E1 15334.376,E2 15334.376} C_VEL
LIN {X 0,Y 397.756,Z 850.018,A -85,B 0,C 180,E1 15333.296,E2 15333.296} C_VEL
LIN {X 0,Y 403.894,Z 827.252,A -85,B 0,C 180,E1 15332.236,E2 15332.236} C_VEL
LIN {X 0,Y 409.005,Z 803.859,A -85,B 0,C 180,E1 15331.394,E2 15331.394} C_VEL
LIN {X 0,Y 413.132,Z 780.688,A -85,B 0,C 180,E1 15330.746,E2 15330.746} C_VEL
LIN {X 0,Y 416.173,Z 755.582,A -85,B 0,C 180,E1 15330.22,E2 15330.22} C_VEL
LIN {X 0,Y 432.44,Z 534.422,A -85,B 0,C 180,E1 15326.598,E2 15326.598} C_VEL
LIN {X 0,Y 425.765,Z 521.335,A -85,B 0,C 180,E1 15324.34,E2 15324.34} C_VEL
LIN {X 0,Y 419.365,Z 509.666,A -85,B 0,C 180,E1 15321.946,E2 15321.946} C_VEL
LIN {X 0,Y 413.828,Z 500.099,A -85,B 0,C 180,E1 15319.624,E2 15319.624} C_VEL
LIN {X 0,Y 408.544,Z 492.288,A -85,B 0,C 180,E1 15317.153,E2 15317.153} C_VEL
LIN {X 0,Y 404.593,Z 486.761,A -85,B 0,C 180,E1 15315.04,E2 15315.04} C_VEL
LIN {X 0,Y 401.658,Z 482.574,A -85,B 0,C 180,E1 15313.24,E2 15313.24} C_VEL
LIN {X 0,Y 397.969,Z 477.456,A -85,B 0,C 180,E1 15310.569,E2 15310.569} C_VEL
LIN {X 0,Y 395.072,Z 473.702,A -85,B 0,C 180,E1 15307.928,E2 15307.928} C_VEL
LIN {X 0,Y 394.278,Z 472.195,A -85,B 0,C 180,E1 15306.992,E2 15306.992} C_VEL
LIN {X 0,Y 390.943,Z 466.591,A -85,B 0,C 180,E1 15298.828,E2 15298.828} C_VEL
LIN {X 0,Y 391.332,Z 468.804,A -85,B 0,C 180,E1 15295.457,E2 15295.457} C_VEL
LIN {X 0,Y 394.595,Z 472.62,A -85,B 0,C 180,E1 15290.225,E2 15290.225} C_VEL
LIN {X 0,Y 397.351,Z 476.896,A -85,B 0,C 180,E1 15287.502,E2 15287.502} C_VEL
LIN {X 0,Y 398.703,Z 478.42,A -85,B 0,C 180,E1 15286.439,E2 15286.439} C_VEL
LIN {X 0,Y 402.767,Z 484.173,A -85,B 0,C 180,E1 15283.634,E2 15283.634} C_VEL
LIN {X 0,Y 406.481,Z 489.377,A -85,B 0,C 180,E1 15281.499,E2 15281.499} C_VEL
LIN {X 0,Y 410.443,Z 495.07,A -85,B 0,C 180,E1 15279.501,E2 15279.501} C_VEL
LIN {X 0,Y 415.829,Z 502.974,A -85,B 0,C 180,E1 15277.111,E2 15277.111} C_VEL
LIN {X 0,Y 423.519,Z 514.987,A -85,B 0,C 180,E1 15274.14,E2 15274.14} C_VEL
LIN {X 0,Y 431.288,Z 527.889,A -85,B 0,C 180,E1 15271.51,E2 15271.51} C_VEL
LIN {X 0,Y 432.587,Z 530.46,A -85,B 0,C 180,E1 15271.087,E2 15271.087} C_VEL
LIN {X 0,Y 416.611,Z 746.198,A -85,B 0,C 180,E1 15267.556,E2 15267.556} C_VEL
LIN {X 0,Y 413.237,Z 772.776,A -85,B 0,C 180,E1 15266.956,E2 15266.956} C_VEL
LIN {X 0,Y 409.644,Z 793.399,A -85,B 0,C 180,E1 15266.332,E2 15266.332} C_VEL
LIN {X 0,Y 404.466,Z 817.349,A -85,B 0,C 180,E1 15265.408,E2 15265.408} C_VEL
LIN {X 0,Y 399.021,Z 837.987,A -85,B 0,C 180,E1 15264.405,E2 15264.405} C_VEL
LIN {X 0,Y 392.484,Z 859.751,A -85,B 0,C 180,E1 15263.125,E2 15263.125} C_VEL
LIN {X 0,Y 385.178,Z 880.634,A -85,B 0,C 180,E1 15261.625,E2 15261.625} C_VEL
LIN {X 0,Y 378.164,Z 898.884,A -85,B 0,C 180,E1 15260.065,E2 15260.065} C_VEL
LIN {X 0,Y 369.204,Z 920.008,A -85,B 0,C 180,E1 15257.907,E2 15257.907} C_VEL
LIN {X 0,Y 361.513,Z 936.692,A -85,B 0,C 180,E1 15255.868,E2 15255.868} C_VEL
LIN {X 0,Y 352.516,Z 955.067,A -85,B 0,C 180,E1 15253.2,E2 15253.2} C_VEL
LIN {X 0,Y 344.576,Z 970.313,A -85,B 0,C 180,E1 15250.542,E2 15250.542} C_VEL
LIN {X 0,Y 336.694,Z 985.124,A -85,B 0,C 180,E1 15247.502,E2 15247.502} C_VEL
LIN {X 0,Y 328.953,Z 999.119,A -85,B 0,C 180,E1 15244.007,E2 15244.007} C_VEL
LIN {X 0,Y 322.348,Z 1011.352,A -85,B 0,C 180,E1 15240.372,E2 15240.372} C_VEL
LIN {X 0,Y 316.58,Z 1022.099,A -85,B 0,C 180,E1 15236.445,E2 15236.445} C_VEL
LIN {X 0,Y 312.039,Z 1031.265,A -85,B 0,C 180,E1 15232.415,E2 15232.415} C_VEL
LIN {X 0,Y 308.405,Z 1039.339,A -85,B 0,C 180,E1 15227.939,E2 15227.939} C_VEL
LIN {X 0,Y 306.264,Z 1045.015,A -85,B 0,C 180,E1 15223.981,E2 15223.981} C_VEL
LIN {X 0,Y 304.773,Z 1050.105,A -85,B 0,C 180,E1 15219.251,E2 15219.251} C_VEL
LIN {X 0,Y 304.21,Z 1053,A -85,B 0,C 180,E1 15215.28,E2 15215.28} C_VEL
LIN {X 0,Y 304.03,Z 1054.698,A -85,B 0,C 180,E1 15211.508,E2 15211.508} C_VEL
LIN {X 0,Y 303.99,Z 1055.394,A -85,B 0,C 180,E1 15207.361,E2 15207.361} C_VEL
LIN {X 0,Y 304.084,Z 1054.663,A -85,B 0,C 180,E1 15203.202,E2 15203.202} C_VEL
LIN {X 0,Y 304.342,Z 1053.049,A -85,B 0,C 180,E1 15199.59,E2 15199.59} C_VEL
LIN {X 0,Y 305.096,Z 1050.156,A -85,B 0,C 180,E1 15195.577,E2 15195.577} C_VEL
LIN {X 0,Y 306.918,Z 1045.034,A -85,B 0,C 180,E1 15190.789,E2 15190.789} C_VEL
LIN {X 0,Y 309.449,Z 1039.309,A -85,B 0,C 180,E1 15186.784,E2 15186.784} C_VEL
LIN {X 0,Y 313.625,Z 1031.117,A -85,B 0,C 180,E1 15182.259,E2 15182.259} C_VEL
LIN {X 0,Y 318.474,Z 1022.276,A -85,B 0,C 180,E1 15178.378,E2 15178.378} C_VEL
LIN {X 0,Y 324.84,Z 1011.42,A -85,B 0,C 180,E1 15174.426,E2 15174.426} C_VEL
LIN {X 0,Y 332.074,Z 999.042,A -85,B 0,C 180,E1 15170.778,E2 15170.778} C_VEL
LIN {X 0,Y 340.062,Z 985.569,A -85,B 0,C 180,E1 15167.447,E2 15167.447} C_VEL
LIN {X 0,Y 348.532,Z 970.629,A -85,B 0,C 180,E1 15164.41,E2 15164.41} C_VEL
LIN {X 0,Y 356.861,Z 955.523,A -85,B 0,C 180,E1 15161.815,E2 15161.815} C_VEL
LIN {X 0,Y 366.378,Z 937.141,A -85,B 0,C 180,E1 15159.189,E2 15159.189} C_VEL
LIN {X 0,Y 374.547,Z 920.273,A -85,B 0,C 180,E1 15157.167,E2 15157.167} C_VEL
LIN {X 0,Y 384.052,Z 898.875,A -85,B 0,C 180,E1 15155.034,E2 15155.034} C_VEL
LIN {X 0,Y 391.16,Z 881.166,A -85,B 0,C 180,E1 15153.558,E2 15153.558} C_VEL
LIN {X 0,Y 399.138,Z 859.19,A -85,B 0,C 180,E1 15152.027,E2 15152.027} C_VEL
LIN {X 0,Y 405.748,Z 837.99,A -85,B 0,C 180,E1 15150.817,E2 15150.817} C_VEL
LIN {X 0,Y 411.995,Z 815.05,A -85,B 0,C 180,E1 15149.745,E2 15149.745} C_VEL
LIN {X 0,Y 412.236,Z 813.969,A -85,B 0,C 180,E1 15149.702,E2 15149.702} C_VEL
LIN {X 0,Y 413.356,Z 806.832,A -85,B 0,C 180,E1 15149.302,E2 15149.302} C_VEL
LIN {X 0,Y 414.24,Z 789.235,A -85,B 0,C 180,E1 15147.956,E2 15147.956} C_VEL
LIN {X 0,Y 415.089,Z 781.926,A -85,B 0,C 180,E1 15147.622,E2 15147.622} C_VEL
LIN {X 0,Y 418.675,Z 758.825,A -85,B 0,C 180,E1 15147.053,E2 15147.053} C_VEL
LIN {X 0,Y 421.397,Z 733.209,A -85,B 0,C 180,E1 15146.578,E2 15146.578} C_VEL
LIN {X 0,Y 436.472,Z 540.091,A -85,B 0,C 180,E1 15143.473,E2 15143.473} C_VEL
LIN {X 0,Y 430.16,Z 529.414,A -85,B 0,C 180,E1 15141.083,E2 15141.083} C_VEL
LIN {X 0,Y 423.64,Z 519,A -85,B 0,C 180,E1 15138.26,E2 15138.26} C_VEL
LIN {X 0,Y 418.868,Z 511.764,A -85,B 0,C 180,E1 15135.862,E2 15135.862} C_VEL
LIN {X 0,Y 415.843,Z 507.313,A -85,B 0,C 180,E1 15134.126,E2 15134.126} C_VEL
LIN {X 0,Y 413.255,Z 503.408,A -85,B 0,C 180,E1 15132.436,E2 15132.436} C_VEL
LIN {X 0,Y 410.054,Z 498.749,A -85,B 0,C 180,E1 15129.97,E2 15129.97} C_VEL
LIN {X 0,Y 407.172,Z 494.337,A -85,B 0,C 180,E1 15127.053,E2 15127.053} C_VEL
LIN {X 0,Y 403.983,Z 488.887,A -85,B 0,C 180,E1 15119.291,E2 15119.291} C_VEL
LIN {X 0,Y 404.263,Z 490.703,A -85,B 0,C 180,E1 15116.313,E2 15116.313} C_VEL
LIN {X 0,Y 407.205,Z 494.378,A -85,B 0,C 180,E1 15111.243,E2 15111.243} C_VEL
LIN {X 0,Y 409.769,Z 498.475,A -85,B 0,C 180,E1 15108.6,E2 15108.6} C_VEL
LIN {X 0,Y 410.93,Z 499.999,A -85,B 0,C 180,E1 15107.636,E2 15107.636} C_VEL
LIN {X 0,Y 414.531,Z 505.26,A -85,B 0,C 180,E1 15105.043,E2 15105.043} C_VEL
LIN {X 0,Y 417.988,Z 510.399,A -85,B 0,C 180,E1 15102.96,E2 15102.96} C_VEL
LIN {X 0,Y 421.29,Z 515.524,A -85,B 0,C 180,E1 15101.205,E2 15101.205} C_VEL
LIN {X 0,Y 428.233,Z 527.953,A -85,B 0,C 180,E1 15097.966,E2 15097.966} C_VEL
LIN {X 0,Y 435.709,Z 542.535,A -85,B 0,C 180,E1 15094.987,E2 15094.987} C_VEL
LIN {X 0,Y 436.342,Z 544.175,A -85,B 0,C 180,E1 15094.739,E2 15094.739} C_VEL
LIN {X 0,Y 419.514,Z 757.283,A -85,B 0,C 180,E1 15091.3,E2 15091.3} C_VEL
LIN {X 0,Y 415.84,Z 784.009,A -85,B 0,C 180,E1 15090.737,E2 15090.737} C_VEL
LIN {X 0,Y 411.668,Z 805.744,A -85,B 0,C 180,E1 15090.138,E2 15090.138} C_VEL
LIN {X 0,Y 405.695,Z 830.577,A -85,B 0,C 180,E1 15089.247,E2 15089.247} C_VEL
LIN {X 0,Y 399.826,Z 850.919,A -85,B 0,C 180,E1 15088.32,E2 15088.32} C_VEL
LIN {X 0,Y 392.489,Z 873.21,A -85,B 0,C 180,E1 15087.079,E2 15087.079} C_VEL
LIN {X 0,Y 384.643,Z 893.826,A -85,B 0,C 180,E1 15085.66,E2 15085.66} C_VEL
LIN {X 0,Y 376.465,Z 913.378,A -85,B 0,C 180,E1 15084.057,E2 15084.057} C_VEL
LIN {X 0,Y 367.131,Z 933.544,A -85,B 0,C 180,E1 15082.042,E2 15082.042} C_VEL
LIN {X 0,Y 358.732,Z 950.377,A -85,B 0,C 180,E1 15080.041,E2 15080.041} C_VEL
LIN {X 0,Y 348.439,Z 969.671,A -85,B 0,C 180,E1 15077.275,E2 15077.275} C_VEL
LIN {X 0,Y 340.417,Z 983.933,A -85,B 0,C 180,E1 15074.825,E2 15074.825} C_VEL
LIN {X 0,Y 331.284,Z 999.705,A -85,B 0,C 180,E1 15071.606,E2 15071.606} C_VEL
LIN {X 0,Y 323.557,Z 1012.659,A -85,B 0,C 180,E1 15068.4,E2 15068.4} C_VEL
LIN {X 0,Y 316.145,Z 1025.308,A -85,B 0,C 180,E1 15064.682,E2 15064.682} C_VEL
LIN {X 0,Y 309.724,Z 1036.399,A -85,B 0,C 180,E1 15060.669,E2 15060.669} C_VEL
LIN {X 0,Y 304.832,Z 1045.506,A -85,B 0,C 180,E1 15056.704,E2 15056.704} C_VEL
LIN {X 0,Y 300.554,Z 1054.364,A -85,B 0,C 180,E1 15051.876,E2 15051.876} C_VEL
LIN {X 0,Y 298.169,Z 1060.337,A -85,B 0,C 180,E1 15047.753,E2 15047.753} C_VEL
LIN {X 0,Y 296.588,Z 1065.714,A -85,B 0,C 180,E1 15042.856,E2 15042.856} C_VEL
LIN {X 0,Y 296.057,Z 1068.802,A -85,B 0,C 180,E1 15038.742,E2 15038.742} C_VEL
LIN {X 0,Y 295.965,Z 1070.558,A -85,B 0,C 180,E1 15035.039,E2 15035.039} C_VEL
LIN {X 0,Y 295.988,Z 1071.34,A -85,B 0,C 180,E1 15031.161,E2 15031.161} C_VEL
LIN {X 0,Y 295.982,Z 1070.949,A -85,B 0,C 180,E1 15027.095,E2 15027.095} C_VEL
LIN {X 0,Y 295.985,Z 1069.219,A -85,B 0,C 180,E1 15023.015,E2 15023.015} C_VEL
LIN {X 0,Y 296.236,Z 1066.514,A -85,B 0,C 180,E1 15019.18,E2 15019.18} C_VEL
LIN {X 0,Y 297.163,Z 1062.133,A -85,B 0,C 180,E1 15014.784,E2 15014.784} C_VEL
LIN {X 0,Y 299.206,Z 1055.636,A -85,B 0,C 180,E1 15010.07,E2 15010.07} C_VEL
LIN {X 0,Y 302.078,Z 1048.532,A -85,B 0,C 180,E1 15005.975,E2 15005.975} C_VEL
LIN {X 0,Y 306.759,Z 1038.581,A -85,B 0,C 180,E1 15001.37,E2 15001.37} C_VEL
LIN {X 0,Y 311.855,Z 1028.689,A -85,B 0,C 180,E1 14997.626,E2 14997.626} C_VEL
LIN {X 0,Y 319.086,Z 1015.375,A -85,B 0,C 180,E1 14993.46,E2 14993.46} C_VEL
LIN {X 0,Y 326.141,Z 1002.551,A -85,B 0,C 180,E1 14990.152,E2 14990.152} C_VEL
LIN {X 0,Y 334.628,Z 987.115,A -85,B 0,C 180,E1 14986.81,E2 14986.81} C_VEL
LIN {X 0,Y 342.594,Z 972.097,A -85,B 0,C 180,E1 14984.113,E2 14984.113} C_VEL
LIN {X 0,Y 351.575,Z 954.674,A -85,B 0,C 180,E1 14981.461,E2 14981.461} C_VEL
LIN {X 0,Y 360.377,Z 936.242,A -85,B 0,C 180,E1 14979.15,E2 14979.15} C_VEL
LIN {X 0,Y 368.441,Z 918.26,A -85,B 0,C 180,E1 14977.242,E2 14977.242} C_VEL
LIN {X 0,Y 377.103,Z 897.095,A -85,B 0,C 180,E1 14975.379,E2 14975.379} C_VEL
LIN {X 0,Y 384.111,Z 878.167,A -85,B 0,C 180,E1 14973.994,E2 14973.994} C_VEL
LIN {X 0,Y 391.773,Z 854.86,A -85,B 0,C 180,E1 14972.583,E2 14972.583} C_VEL
LIN {X 0,Y 397.76,Z 833.621,A -85,B 0,C 180,E1 14971.551,E2 14971.551} C_VEL
LIN {X 0,Y 403.533,Z 809.715,A -85,B 0,C 180,E1 14970.622,E2 14970.622} C_VEL
LIN {X 0,Y 407.972,Z 786.308,A -85,B 0,C 180,E1 14969.936,E2 14969.936} C_VEL
LIN {X 0,Y 411.49,Z 761.682,A -85,B 0,C 180,E1 14969.379,E2 14969.379} C_VEL
LIN {X 0,Y 415.66,Z 708.814,A -85,B 0,C 180,E1 14968.482,E2 14968.482} C_VEL
LIN {X 0,Y 428.389,Z 538.48,A -85,B 0,C 180,E1 14965.697,E2 14965.697} C_VEL
LIN {X 0,Y 422.76,Z 527.263,A -85,B 0,C 180,E1 14963.708,E2 14963.708} C_VEL
LIN {X 0,Y 416.946,Z 516.392,A -85,B 0,C 180,E1 14961.452,E2 14961.452} C_VEL
LIN {X 0,Y 411.771,Z 507.237,A -85,B 0,C 180,E1 14959.21,E2 14959.21} C_VEL
LIN {X 0,Y 406.611,Z 499.485,A -85,B 0,C 180,E1 14956.721,E2 14956.721} C_VEL
LIN {X 0,Y 402.77,Z 493.992,A -85,B 0,C 180,E1 14954.595,E2 14954.595} C_VEL
LIN {X 0,Y 400.136,Z 490.146,A -85,B 0,C 180,E1 14952.924,E2 14952.924} C_VEL
LIN {X 0,Y 396.634,Z 485.178,A -85,B 0,C 180,E1 14950.311,E2 14950.311} C_VEL
LIN {X 0,Y 393.764,Z 481.254,A -85,B 0,C 180,E1 14947.588,E2 14947.588} C_VEL
LIN {X 0,Y 393.175,Z 480.083,A -85,B 0,C 180,E1 14946.865,E2 14946.865} C_VEL
LIN {X 0,Y 389.968,Z 474.534,A -85,B 0,C 180,E1 14938.825,E2 14938.825} C_VEL
LIN {X 0,Y 390.545,Z 477.299,A -85,B 0,C 180,E1 14934.859,E2 14934.859} C_VEL
LIN {X 0,Y 393.421,Z 480.441,A -85,B 0,C 180,E1 14930.425,E2 14930.425} C_VEL
LIN {X 0,Y 396.332,Z 484.908,A -85,B 0,C 180,E1 14927.513,E2 14927.513} C_VEL
LIN {X 0,Y 397.53,Z 486.454,A -85,B 0,C 180,E1 14926.546,E2 14926.546} C_VEL
LIN {X 0,Y 401.23,Z 491.726,A -85,B 0,C 180,E1 14923.941,E2 14923.941} C_VEL
LIN {X 0,Y 404.987,Z 497.134,A -85,B 0,C 180,E1 14921.726,E2 14921.726} C_VEL
LIN {X 0,Y 408.822,Z 502.749,A -85,B 0,C 180,E1 14919.752,E2 14919.752} C_VEL
LIN {X 0,Y 414.357,Z 511.11,A -85,B 0,C 180,E1 14917.25,E2 14917.25} C_VEL
LIN {X 0,Y 421.363,Z 522.322,A -85,B 0,C 180,E1 14914.488,E2 14914.488} C_VEL
LIN {X 0,Y 428.604,Z 534.588,A -85,B 0,C 180,E1 14911.97,E2 14911.97} C_VEL
LIN {X 0,Y 412.497,Z 746.49,A -85,B 0,C 180,E1 14908.504,E2 14908.504} C_VEL
LIN {X 0,Y 409.037,Z 773.102,A -85,B 0,C 180,E1 14907.905,E2 14907.905} C_VEL
LIN {X 0,Y 405.349,Z 793.792,A -85,B 0,C 180,E1 14907.28,E2 14907.28} C_VEL
LIN {X 0,Y 399.987,Z 817.951,A -85,B 0,C 180,E1 14906.35,E2 14906.35} C_VEL
LIN {X 0,Y 394.419,Z 838.544,A -85,B 0,C 180,E1 14905.35,E2 14905.35} C_VEL
LIN {X 0,Y 387.513,Z 860.948,A -85,B 0,C 180,E1 14904.029,E2 14904.029} C_VEL
LIN {X 0,Y 379.937,Z 881.899,A -85,B 0,C 180,E1 14902.51,E2 14902.51} C_VEL
LIN {X 0,Y 372.171,Z 901.502,A -85,B 0,C 180,E1 14900.814,E2 14900.814} C_VEL
LIN {X 0,Y 363.281,Z 921.613,A -85,B 0,C 180,E1 14898.712,E2 14898.712} C_VEL
LIN {X 0,Y 355.136,Z 938.722,A -85,B 0,C 180,E1 14896.586,E2 14896.586} C_VEL
LIN {X 0,Y 345.986,Z 956.649,A -85,B 0,C 180,E1 14893.915,E2 14893.915} C_VEL
LIN {X 0,Y 337.988,Z 971.495,A -85,B 0,C 180,E1 14891.278,E2 14891.278} C_VEL
LIN {X 0,Y 329.044,Z 987.524,A -85,B 0,C 180,E1 14887.867,E2 14887.867} C_VEL
LIN {X 0,Y 321.873,Z 1000.061,A -85,B 0,C 180,E1 14884.645,E2 14884.645} C_VEL
LIN {X 0,Y 314.734,Z 1012.678,A -85,B 0,C 180,E1 14880.763,E2 14880.763} C_VEL
LIN {X 0,Y 309.057,Z 1022.838,A -85,B 0,C 180,E1 14876.932,E2 14876.932} C_VEL
LIN {X 0,Y 304.159,Z 1032.324,A -85,B 0,C 180,E1 14872.62,E2 14872.62} C_VEL
LIN {X 0,Y 300.562,Z 1039.899,A -85,B 0,C 180,E1 14868.223,E2 14868.223} C_VEL
LIN {X 0,Y 298.255,Z 1045.767,A -85,B 0,C 180,E1 14863.968,E2 14863.968} C_VEL
LIN {X 0,Y 296.76,Z 1050.611,A -85,B 0,C 180,E1 14859.168,E2 14859.168} C_VEL
LIN {X 0,Y 296.211,Z 1053.343,A -85,B 0,C 180,E1 14855.229,E2 14855.229} C_VEL
LIN {X 0,Y 296.025,Z 1055.073,A -85,B 0,C 180,E1 14851.111,E2 14851.111} C_VEL
LIN {X 0,Y 295.998,Z 1055.538,A -85,B 0,C 180,E1 14846.708,E2 14846.708} C_VEL
LIN {X 0,Y 296.102,Z 1054.801,A -85,B 0,C 180,E1 14842.822,E2 14842.822} C_VEL
LIN {X 0,Y 296.423,Z 1053.071,A -85,B 0,C 180,E1 14838.993,E2 14838.993} C_VEL
LIN {X 0,Y 297.44,Z 1049.704,A -85,B 0,C 180,E1 14834.399,E2 14834.399} C_VEL
LIN {X 0,Y 299.388,Z 1044.714,A -85,B 0,C 180,E1 14829.879,E2 14829.879} C_VEL
LIN {X 0,Y 302.353,Z 1038.587,A -85,B 0,C 180,E1 14825.583,E2 14825.583} C_VEL
LIN {X 0,Y 306.965,Z 1030.074,A -85,B 0,C 180,E1 14820.965,E2 14820.965} C_VEL
LIN {X 0,Y 312.001,Z 1021.516,A -85,B 0,C 180,E1 14817.207,E2 14817.207} C_VEL
LIN {X 0,Y 319.464,Z 1009.275,A -85,B 0,C 180,E1 14812.838,E2 14812.838} C_VEL
LIN {X 0,Y 326.479,Z 997.901,A -85,B 0,C 180,E1 14809.513,E2 14809.513} C_VEL
LIN {X 0,Y 335.765,Z 982.636,A -85,B 0,C 180,E1 14805.826,E2 14805.826} C_VEL
LIN {X 0,Y 343.775,Z 969.032,A -85,B 0,C 180,E1 14803.11,E2 14803.11} C_VEL
LIN {X 0,Y 353.545,Z 951.748,A -85,B 0,C 180,E1 14800.217,E2 14800.217} C_VEL
LIN {X 0,Y 362.382,Z 934.969,A -85,B 0,C 180,E1 14797.895,E2 14797.895} C_VEL
LIN {X 0,Y 371.769,Z 915.98,A -85,B 0,C 180,E1 14795.684,E2 14795.684} C_VEL
LIN {X 0,Y 380.361,Z 896.66,A -85,B 0,C 180,E1 14793.829,E2 14793.829} C_VEL
LIN {X 0,Y 388.68,Z 876.258,A -85,B 0,C 180,E1 14792.182,E2 14792.182} C_VEL
LIN {X 0,Y 396.269,Z 854.919,A -85,B 0,C 180,E1 14790.776,E2 14790.776} C_VEL
LIN {X 0,Y 402.897,Z 833.756,A -85,B 0,C 180,E1 14789.613,E2 14789.613} C_VEL
LIN {X 0,Y 409.117,Z 810.129,A -85,B 0,C 180,E1 14788.574,E2 14788.574} C_VEL
LIN {X 0,Y 413.805,Z 788.624,A -85,B 0,C 180,E1 14787.825,E2 14787.825} C_VEL
LIN {X 0,Y 415.089,Z 781.926,A -85,B 0,C 180,E1 14787.622,E2 14787.622} C_VEL
LIN {X 0,Y 415.873,Z 774.544,A -85,B 0,C 180,E1 14787.306,E2 14787.306} C_VEL
LIN {X 0,Y 415.898,Z 755.236,A -85,B 0,C 180,E1 14786.092,E2 14786.092} C_VEL
LIN {X 0,Y 416.266,Z 748.79,A -85,B 0,C 180,E1 14785.874,E2 14785.874} C_VEL
LIN {X 0,Y 422.531,Z 672.842,A -85,B 0,C 180,E1 14784.631,E2 14784.631} C_VEL
LIN {X 0,Y 432.857,Z 544.806,A -85,B 0,C 180,E1 14782.587,E2 14782.587} C_VEL
LIN {X 0,Y 425.931,Z 532.993,A -85,B 0,C 180,E1 14779.794,E2 14779.794} C_VEL
LIN {X 0,Y 420.009,Z 523.559,A -85,B 0,C 180,E1 14777.027,E2 14777.027} C_VEL
LIN {X 0,Y 415.196,Z 516.036,A -85,B 0,C 180,E1 14774.362,E2 14774.362} C_VEL
LIN {X 0,Y 411.681,Z 510.855,A -85,B 0,C 180,E1 14772.057,E2 14772.057} C_VEL
LIN {X 0,Y 408.914,Z 506.631,A -85,B 0,C 180,E1 14769.856,E2 14769.856} C_VEL
LIN {X 0,Y 406.016,Z 502.153,A -85,B 0,C 180,E1 14766.86,E2 14766.86} C_VEL
LIN {X 0,Y 403.007,Z 496.84,A -85,B 0,C 180,E1 14759.289,E2 14759.289} C_VEL
LIN {X 0,Y 403.667,Z 499.483,A -85,B 0,C 180,E1 14755.169,E2 14755.169} C_VEL
LIN {X 0,Y 406.05,Z 502.204,A -85,B 0,C 180,E1 14751.432,E2 14751.432} C_VEL
LIN {X 0,Y 408.637,Z 506.362,A -85,B 0,C 180,E1 14748.711,E2 14748.711} C_VEL
LIN {X 0,Y 409.689,Z 507.854,A -85,B 0,C 180,E1 14747.812,E2 14747.812} C_VEL
LIN {X 0,Y 413.229,Z 513.15,A -85,B 0,C 180,E1 14745.21,E2 14745.21} C_VEL
LIN {X 0,Y 416.523,Z 518.143,A -85,B 0,C 180,E1 14743.186,E2 14743.186} C_VEL
LIN {X 0,Y 419.575,Z 523.022,A -85,B 0,C 180,E1 14741.521,E2 14741.521} C_VEL
LIN {X 0,Y 426.109,Z 535.032,A -85,B 0,C 180,E1 14738.382,E2 14738.382} C_VEL
LIN {X 0,Y 432.734,Z 548.357,A -85,B 0,C 180,E1 14735.639,E2 14735.639} C_VEL
LIN {X 0,Y 415.839,Z 757.029,A -85,B 0,C 180,E1 14732.281,E2 14732.281} C_VEL
LIN {X 0,Y 412.084,Z 783.835,A -85,B 0,C 180,E1 14731.72,E2 14731.72} C_VEL
LIN {X 0,Y 407.847,Z 805.498,A -85,B 0,C 180,E1 14731.129,E2 14731.129} C_VEL
LIN {X 0,Y 401.88,Z 829.898,A -85,B 0,C 180,E1 14730.264,E2 14730.264} C_VEL
LIN {X 0,Y 396.158,Z 849.397,A -85,B 0,C 180,E1 14729.392,E2 14729.392} C_VEL
LIN {X 0,Y 389.177,Z 870.341,A -85,B 0,C 180,E1 14728.257,E2 14728.257} C_VEL
LIN {X 0,Y 380.702,Z 892.427,A -85,B 0,C 180,E1 14726.774,E2 14726.774} C_VEL
LIN {X 0,Y 372.817,Z 910.888,A -85,B 0,C 180,E1 14725.288,E2 14725.288} C_VEL
LIN {X 0,Y 362.773,Z 932.271,A -85,B 0,C 180,E1 14723.196,E2 14723.196} C_VEL
LIN {X 0,Y 354.101,Z 949.195,A -85,B 0,C 180,E1 14721.201,E2 14721.201} C_VEL
LIN {X 0,Y 343.991,Z 967.716,A -85,B 0,C 180,E1 14718.585,E2 14718.585} C_VEL
LIN {X 0,Y 334.973,Z 983.222,A -85,B 0,C 180,E1 14715.932,E2 14715.932} C_VEL
LIN {X 0,Y 325.607,Z 998.873,A -85,B 0,C 180,E1 14712.739,E2 14712.739} C_VEL
LIN {X 0,Y 317.11,Z 1012.523,A -85,B 0,C 180,E1 14709.33,E2 14709.33} C_VEL
LIN {X 0,Y 309.394,Z 1025.113,A -85,B 0,C 180,E1 14705.571,E2 14705.571} C_VEL
LIN {X 0,Y 302.628,Z 1036.239,A -85,B 0,C 180,E1 14701.469,E2 14701.469} C_VEL
LIN {X 0,Y 297.469,Z 1045.339,A -85,B 0,C 180,E1 14697.42,E2 14697.42} C_VEL
LIN {X 0,Y 293.076,Z 1053.875,A -85,B 0,C 180,E1 14692.676,E2 14692.676} C_VEL
LIN {X 0,Y 290.474,Z 1059.872,A -85,B 0,C 180,E1 14688.463,E2 14688.463} C_VEL
LIN {X 0,Y 288.747,Z 1065.188,A -85,B 0,C 180,E1 14683.62,E2 14683.62} C_VEL
LIN {X 0,Y 288.079,Z 1068.483,A -85,B 0,C 180,E1 14679.187,E2 14679.187} C_VEL
LIN {X 0,Y 287.967,Z 1070.282,A -85,B 0,C 180,E1 14675.379,E2 14675.379} C_VEL
LIN {X 0,Y 287.985,Z 1071.082,A -85,B 0,C 180,E1 14671.592,E2 14671.592} C_VEL
LIN {X 0,Y 287.985,Z 1070.834,A -85,B 0,C 180,E1 14667.413,E2 14667.413} C_VEL
LIN {X 0,Y 287.986,Z 1069.107,A -85,B 0,C 180,E1 14663.02,E2 14663.02} C_VEL
LIN {X 0,Y 288.257,Z 1066.378,A -85,B 0,C 180,E1 14659.002,E2 14659.002} C_VEL
LIN {X 0,Y 289.162,Z 1062.293,A -85,B 0,C 180,E1 14654.744,E2 14654.744} C_VEL
LIN {X 0,Y 291.363,Z 1055.687,A -85,B 0,C 180,E1 14649.72,E2 14649.72} C_VEL
LIN {X 0,Y 294.375,Z 1048.627,A -85,B 0,C 180,E1 14645.519,E2 14645.519} C_VEL
LIN {X 0,Y 299.508,Z 1038.299,A -85,B 0,C 180,E1 14640.61,E2 14640.61} C_VEL
LIN {X 0,Y 304.87,Z 1028.398,A -85,B 0,C 180,E1 14636.79,E2 14636.79} C_VEL
LIN {X 0,Y 312.45,Z 1015.068,A -85,B 0,C 180,E1 14632.553,E2 14632.553} C_VEL
LIN {X 0,Y 319.807,Z 1002.235,A -85,B 0,C 180,E1 14629.198,E2 14629.198} C_VEL
LIN {X 0,Y 328.611,Z 986.823,A -85,B 0,C 180,E1 14625.83,E2 14625.83} C_VEL
LIN {X 0,Y 337.253,Z 971.088,A -85,B 0,C 180,E1 14622.993,E2 14622.993} C_VEL
LIN {X 0,Y 346.72,Z 953.222,A -85,B 0,C 180,E1 14620.29,E2 14620.29} C_VEL
LIN {X 0,Y 355.534,Z 935.243,A -85,B 0,C 180,E1 14618.051,E2 14618.051} C_VEL
LIN {X 0,Y 364.125,Z 916.576,A -85,B 0,C 180,E1 14616.086,E2 14616.086} C_VEL
LIN {X 0,Y 372.799,Z 895.718,A -85,B 0,C 180,E1 14614.281,E2 14614.281} C_VEL
LIN {X 0,Y 379.948,Z 876.799,A -85,B 0,C 180,E1 14612.913,E2 14612.913} C_VEL
LIN {X 0,Y 387.699,Z 853.539,A -85,B 0,C 180,E1 14611.529,E2 14611.529} C_VEL
LIN {X 0,Y 393.582,Z 833.06,A -85,B 0,C 180,E1 14610.546,E2 14610.546} C_VEL
LIN {X 0,Y 399.52,Z 808.81,A -85,B 0,C 180,E1 14609.617,E2 14609.617} C_VEL
LIN {X 0,Y 403.96,Z 785.8,A -85,B 0,C 180,E1 14608.951,E2 14608.951} C_VEL
LIN {X 0,Y 407.539,Z 760.984,A -85,B 0,C 180,E1 14608.395,E2 14608.395} C_VEL
LIN {X 0,Y 412.003,Z 705.545,A -85,B 0,C 180,E1 14607.459,E2 14607.459} C_VEL
LIN {X 0,Y 424.479,Z 542.553,A -85,B 0,C 180,E1 14604.79,E2 14604.79} C_VEL
LIN {X 0,Y 417.996,Z 529.525,A -85,B 0,C 180,E1 14602.355,E2 14602.355} C_VEL
LIN {X 0,Y 411.257,Z 516.965,A -85,B 0,C 180,E1 14599.493,E2 14599.493} C_VEL
LIN {X 0,Y 407.07,Z 510.274,A -85,B 0,C 180,E1 14597.512,E2 14597.512} C_VEL
LIN {X 0,Y 401.903,Z 502.437,A -85,B 0,C 180,E1 14594.7,E2 14594.7} C_VEL
LIN {X 0,Y 398.522,Z 497.598,A -85,B 0,C 180,E1 14592.535,E2 14592.535} C_VEL
LIN {X 0,Y 395.306,Z 492.897,A -85,B 0,C 180,E1 14590.051,E2 14590.051} C_VEL
LIN {X 0,Y 392.528,Z 488.937,A -85,B 0,C 180,E1 14587.317,E2 14587.317} C_VEL
LIN {X 0,Y 391.947,Z 487.896,A -85,B 0,C 180,E1 14586.592,E2 14586.592} C_VEL
LIN {X 0,Y 388.991,Z 482.499,A -85,B 0,C 180,E1 14578.674,E2 14578.674} C_VEL
LIN {X 0,Y 392.262,Z 488.286,A -85,B 0,C 180,E1 14570.611,E2 14570.611} C_VEL
LIN {X 0,Y 395.071,Z 492.677,A -85,B 0,C 180,E1 14567.725,E2 14567.725} C_VEL
LIN {X 0,Y 396.19,Z 494.16,A -85,B 0,C 180,E1 14566.797,E2 14566.797} C_VEL
LIN {X 0,Y 399.81,Z 499.457,A -85,B 0,C 180,E1 14564.181,E2 14564.181} C_VEL
LIN {X 0,Y 403.5,Z 504.884,A -85,B 0,C 180,E1 14561.955,E2 14561.955} C_VEL
LIN {X 0,Y 408.402,Z 512.099,A -85,B 0,C 180,E1 14559.431,E2 14559.431} C_VEL
LIN {X 0,Y 414.685,Z 522.176,A -85,B 0,C 180,E1 14556.631,E2 14556.631} C_VEL
LIN {X 0,Y 421.744,Z 533.898,A -85,B 0,C 180,E1 14553.909,E2 14553.909} C_VEL
LIN {X 0,Y 424.679,Z 539.346,A -85,B 0,C 180,E1 14552.859,E2 14552.859} C_VEL
LIN {X 0,Y 408.507,Z 746.677,A -85,B 0,C 180,E1 14549.473,E2 14549.473} C_VEL
LIN {X 0,Y 404.973,Z 773.299,A -85,B 0,C 180,E1 14548.877,E2 14548.877} C_VEL
LIN {X 0,Y 401.214,Z 793.942,A -85,B 0,C 180,E1 14548.258,E2 14548.258} C_VEL
LIN {X 0,Y 395.957,Z 817.28,A -85,B 0,C 180,E1 14547.37,E2 14547.37} C_VEL
LIN {X 0,Y 389.927,Z 839.1,A -85,B 0,C 180,E1 14546.316,E2 14546.316} C_VEL
LIN {X 0,Y 382.84,Z 861.502,A -85,B 0,C 180,E1 14544.996,E2 14544.996} C_VEL
LIN {X 0,Y 375.101,Z 882.36,A -85,B 0,C 180,E1 14543.484,E2 14543.484} C_VEL
LIN {X 0,Y 366.838,Z 902.668,A -85,B 0,C 180,E1 14541.721,E2 14541.721} C_VEL
LIN {X 0,Y 358.002,Z 922.016,A -85,B 0,C 180,E1 14539.683,E2 14539.683} C_VEL
LIN {X 0,Y 349.622,Z 939.11,A -85,B 0,C 180,E1 14537.549,E2 14537.549} C_VEL
LIN {X 0,Y 340.182,Z 957.009,A -85,B 0,C 180,E1 14534.864,E2 14534.864} C_VEL
LIN {X 0,Y 331.75,Z 972.148,A -85,B 0,C 180,E1 14532.145,E2 14532.145} C_VEL
LIN {X 0,Y 322.237,Z 988.539,A -85,B 0,C 180,E1 14528.587,E2 14528.587} C_VEL
LIN {X 0,Y 314.833,Z 1001.002,A -85,B 0,C 180,E1 14525.311,E2 14525.311} C_VEL
LIN {X 0,Y 306.895,Z 1014.378,A -85,B 0,C 180,E1 14521.032,E2 14521.032} C_VEL
LIN {X 0,Y 301.308,Z 1024.027,A -85,B 0,C 180,E1 14517.255,E2 14517.255} C_VEL
LIN {X 0,Y 295.904,Z 1033.979,A -85,B 0,C 180,E1 14512.448,E2 14512.448} C_VEL
LIN {X 0,Y 292.592,Z 1040.756,A -85,B 0,C 180,E1 14508.324,E2 14508.324} C_VEL
LIN {X 0,Y 290.083,Z 1046.948,A -85,B 0,C 180,E1 14503.556,E2 14503.556} C_VEL
LIN {X 0,Y 288.764,Z 1051.05,A -85,B 0,C 180,E1 14499.165,E2 14499.165} C_VEL
LIN {X 0,Y 288.211,Z 1053.685,A -85,B 0,C 180,E1 14495.175,E2 14495.175} C_VEL
LIN {X 0,Y 288.019,Z 1055.463,A -85,B 0,C 180,E1 14490.597,E2 14490.597} C_VEL
LIN {X 0,Y 288.005,Z 1055.705,A -85,B 0,C 180,E1 14486.218,E2 14486.218} C_VEL
LIN {X 0,Y 288.123,Z 1054.94,A -85,B 0,C 180,E1 14482.422,E2 14482.422} C_VEL
LIN {X 0,Y 288.513,Z 1053.115,A -85,B 0,C 180,E1 14478.404,E2 14478.404} C_VEL
LIN {X 0,Y 289.793,Z 1049.283,A -85,B 0,C 180,E1 14473.359,E2 14473.359} C_VEL
LIN {X 0,Y 291.925,Z 1044.394,A -85,B 0,C 180,E1 14468.922,E2 14468.922} C_VEL
LIN {X 0,Y 295.571,Z 1037.495,A -85,B 0,C 180,E1 14464.126,E2 14464.126} C_VEL
LIN {X 0,Y 300.228,Z 1029.43,A -85,B 0,C 180,E1 14459.808,E2 14459.808} C_VEL
LIN {X 0,Y 306.254,Z 1019.849,A -85,B 0,C 180,E1 14455.61,E2 14455.61} C_VEL
LIN {X 0,Y 313.616,Z 1008.268,A -85,B 0,C 180,E1 14451.559,E2 14451.559} C_VEL
LIN {X 0,Y 321.511,Z 996.063,A -85,B 0,C 180,E1 14448.012,E2 14448.012} C_VEL
LIN {X 0,Y 330.651,Z 981.473,A -85,B 0,C 180,E1 14444.553,E2 14444.553} C_VEL
LIN {X 0,Y 339.237,Z 967.4,A -85,B 0,C 180,E1 14441.769,E2 14441.769} C_VEL
LIN {X 0,Y 349.394,Z 949.786,A -85,B 0,C 180,E1 14438.885,E2 14438.885} C_VEL
LIN {X 0,Y 358.057,Z 933.776,A -85,B 0,C 180,E1 14436.699,E2 14436.699} C_VEL
LIN {X 0,Y 368.287,Z 913.322,A -85,B 0,C 180,E1 14434.376,E2 14434.376} C_VEL
LIN {X 0,Y 376.198,Z 895.916,A -85,B 0,C 180,E1 14432.731,E2 14432.731} C_VEL
LIN {X 0,Y 384.849,Z 875.072,A -85,B 0,C 180,E1 14431.074,E2 14431.074} C_VEL
LIN {X 0,Y 392.189,Z 854.792,A -85,B 0,C 180,E1 14429.755,E2 14429.755} C_VEL
LIN {X 0,Y 398.983,Z 833.545,A -85,B 0,C 180,E1 14428.598,E2 14428.598} C_VEL
LIN {X 0,Y 405.258,Z 810.118,A -85,B 0,C 180,E1 14427.579,E2 14427.579} C_VEL
LIN {X 0,Y 410.097,Z 788.311,A -85,B 0,C 180,E1 14426.827,E2 14426.827} C_VEL
LIN {X 0,Y 414.512,Z 762.333,A -85,B 0,C 180,E1 14426.15,E2 14426.15} C_VEL
LIN {X 0,Y 416.266,Z 748.79,A -85,B 0,C 180,E1 14425.874,E2 14425.874} C_VEL
LIN {X 0,Y 416.56,Z 741.255,A -85,B 0,C 180,E1 14425.616,E2 14425.616} C_VEL
LIN {X 0,Y 415.51,Z 721.595,A -85,B 0,C 180,E1 14424.516,E2 14424.516} C_VEL
LIN {X 0,Y 415.705,Z 715.097,A -85,B 0,C 180,E1 14424.319,E2 14424.319} C_VEL
LIN {X 0,Y 429.308,Z 549.524,A -85,B 0,C 180,E1 14421.674,E2 14421.674} C_VEL
LIN {X 0,Y 423.035,Z 538.788,A -85,B 0,C 180,E1 14419.013,E2 14419.013} C_VEL
LIN {X 0,Y 417.915,Z 530.42,A -85,B 0,C 180,E1 14416.506,E2 14416.506} C_VEL
LIN {X 0,Y 413.316,Z 523.144,A -85,B 0,C 180,E1 14413.857,E2 14413.857} C_VEL
LIN {X 0,Y 410.314,Z 518.541,A -85,B 0,C 180,E1 14411.812,E2 14411.812} C_VEL
LIN {X 0,Y 407.612,Z 514.346,A -85,B 0,C 180,E1 14409.602,E2 14409.602} C_VEL
LIN {X 0,Y 404.535,Z 509.534,A -85,B 0,C 180,E1 14406.244,E2 14406.244} C_VEL
LIN {X 0,Y 402.031,Z 504.781,A -85,B 0,C 180,E1 14399.145,E2 14399.145} C_VEL
LIN {X 0,Y 404.899,Z 510.028,A -85,B 0,C 180,E1 14391.622,E2 14391.622} C_VEL
LIN {X 0,Y 407.506,Z 514.248,A -85,B 0,C 180,E1 14388.823,E2 14388.823} C_VEL
LIN {X 0,Y 409.195,Z 517.002,A -85,B 0,C 180,E1 14387.367,E2 14387.367} C_VEL
LIN {X 0,Y 411.637,Z 520.527,A -85,B 0,C 180,E1 14385.583,E2 14385.583} C_VEL
LIN {X 0,Y 415.064,Z 525.883,A -85,B 0,C 180,E1 14383.413,E2 14383.413} C_VEL
LIN {X 0,Y 417.873,Z 530.518,A -85,B 0,C 180,E1 14381.84,E2 14381.84} C_VEL
LIN {X 0,Y 423.983,Z 542.072,A -85,B 0,C 180,E1 14378.813,E2 14378.813} C_VEL
LIN {X 0,Y 429.212,Z 552.824,A -85,B 0,C 180,E1 14376.55,E2 14376.55} C_VEL
LIN {X 0,Y 412.278,Z 756.881,A -85,B 0,C 180,E1 14373.276,E2 14373.276} C_VEL
LIN {X 0,Y 408.476,Z 783.53,A -85,B 0,C 180,E1 14372.723,E2 14372.723} C_VEL
LIN {X 0,Y 404.178,Z 805.123,A -85,B 0,C 180,E1 14372.141,E2 14372.141} C_VEL
LIN {X 0,Y 397.959,Z 830.029,A -85,B 0,C 180,E1 14371.268,E2 14371.268} C_VEL
LIN {X 0,Y 392.12,Z 849.486,A -85,B 0,C 180,E1 14370.405,E2 14370.405} C_VEL
LIN {X 0,Y 384.643,Z 871.4,A -85,B 0,C 180,E1 14369.221,E2 14369.221} C_VEL
LIN {X 0,Y 375.982,Z 893.24,A -85,B 0,C 180,E1 14367.746,E2 14367.746} C_VEL
LIN {X 0,Y 367.268,Z 913.073,A -85,B 0,C 180,E1 14366.136,E2 14366.136} C_VEL
LIN {X 0,Y 357.356,Z 933.354,A -85,B 0,C 180,E1 14364.117,E2 14364.117} C_VEL
LIN {X 0,Y 348.137,Z 950.795,A -85,B 0,C 180,E1 14362.036,E2 14362.036} C_VEL
LIN {X 0,Y 337.465,Z 969.534,A -85,B 0,C 180,E1 14359.319,E2 14359.319} C_VEL
LIN {X 0,Y 328.891,Z 983.777,A -85,B 0,C 180,E1 14356.839,E2 14356.839} C_VEL
LIN {X 0,Y 319.119,Z 999.452,A -85,B 0,C 180,E1 14353.577,E2 14353.577} C_VEL
LIN {X 0,Y 310.753,Z 1012.387,A -85,B 0,C 180,E1 14350.297,E2 14350.297} C_VEL
LIN {X 0,Y 302.691,Z 1024.969,A -85,B 0,C 180,E1 14346.484,E2 14346.484} C_VEL
LIN {X 0,Y 295.454,Z 1036.304,A -85,B 0,C 180,E1 14342.214,E2 14342.214} C_VEL
LIN {X 0,Y 289.701,Z 1045.994,A -85,B 0,C 180,E1 14337.772,E2 14337.772} C_VEL
LIN {X 0,Y 285.17,Z 1054.313,A -85,B 0,C 180,E1 14332.905,E2 14332.905} C_VEL
LIN {X 0,Y 282.411,Z 1060.425,A -85,B 0,C 180,E1 14328.401,E2 14328.401} C_VEL
LIN {X 0,Y 280.642,Z 1065.65,A -85,B 0,C 180,E1 14323.181,E2 14323.181} C_VEL
LIN {X 0,Y 280.071,Z 1068.517,A -85,B 0,C 180,E1 14319.038,E2 14319.038} C_VEL
LIN {X 0,Y 279.968,Z 1070.217,A -85,B 0,C 180,E1 14315.123,E2 14315.123} C_VEL
LIN {X 0,Y 279.997,Z 1070.97,A -85,B 0,C 180,E1 14310.783,E2 14310.783} C_VEL
LIN {X 0,Y 279.979,Z 1070.365,A -85,B 0,C 180,E1 14306.519,E2 14306.519} C_VEL
LIN {X 0,Y 280.001,Z 1068.643,A -85,B 0,C 180,E1 14302.407,E2 14302.407} C_VEL
LIN {X 0,Y 280.361,Z 1065.813,A -85,B 0,C 180,E1 14298.271,E2 14298.271} C_VEL
LIN {X 0,Y 281.638,Z 1060.925,A -85,B 0,C 180,E1 14293.287,E2 14293.287} C_VEL
LIN {X 0,Y 283.905,Z 1054.806,A -85,B 0,C 180,E1 14288.73,E2 14288.73} C_VEL
LIN {X 0,Y 287.616,Z 1046.913,A -85,B 0,C 180,E1 14284.021,E2 14284.021} C_VEL
LIN {X 0,Y 292.82,Z 1037.08,A -85,B 0,C 180,E1 14279.417,E2 14279.417} C_VEL
LIN {X 0,Y 298.908,Z 1026.533,A -85,B 0,C 180,E1 14275.342,E2 14275.342} C_VEL
LIN {X 0,Y 306.651,Z 1013.468,A -85,B 0,C 180,E1 14271.241,E2 14271.241} C_VEL
LIN {X 0,Y 314.436,Z 1000.495,A -85,B 0,C 180,E1 14267.858,E2 14267.858} C_VEL
LIN {X 0,Y 323.692,Z 984.772,A -85,B 0,C 180,E1 14264.475,E2 14264.475} C_VEL
LIN {X 0,Y 331.827,Z 970.468,A -85,B 0,C 180,E1 14261.903,E2 14261.903} C_VEL
LIN {X 0,Y 341.415,Z 952.907,A -85,B 0,C 180,E1 14259.242,E2 14259.242} C_VEL
LIN {X 0,Y 350.523,Z 934.858,A -85,B 0,C 180,E1 14256.992,E2 14256.992} C_VEL
LIN {X 0,Y 359.801,Z 915.22,A -85,B 0,C 180,E1 14254.935,E2 14254.935} C_VEL
LIN {X 0,Y 368.539,Z 894.582,A -85,B 0,C 180,E1 14253.176,E2 14253.176} C_VEL
LIN {X 0,Y 376.276,Z 874.492,A -85,B 0,C 180,E1 14251.746,E2 14251.746} C_VEL
LIN {X 0,Y 383.865,Z 851.878,A -85,B 0,C 180,E1 14250.437,E2 14250.437} C_VEL
LIN {X 0,Y 389.529,Z 832.498,A -85,B 0,C 180,E1 14249.52,E2 14249.52} C_VEL
LIN {X 0,Y 395.621,Z 807.974,A -85,B 0,C 180,E1 14248.594,E2 14248.594} C_VEL
LIN {X 0,Y 400.052,Z 785.373,A -85,B 0,C 180,E1 14247.948,E2 14247.948} C_VEL
LIN {X 0,Y 403.701,Z 760.378,A -85,B 0,C 180,E1 14247.395,E2 14247.395} C_VEL
LIN {X 0,Y 408.476,Z 702.307,A -85,B 0,C 180,E1 14246.418,E2 14246.418} C_VEL
LIN {X 0,Y 420.683,Z 546.685,A -85,B 0,C 180,E1 14243.87,E2 14243.87} C_VEL
LIN {X 0,Y 413.283,Z 531.787,A -85,B 0,C 180,E1 14240.908,E2 14240.908} C_VEL
LIN {X 0,Y 407.708,Z 521.486,A -85,B 0,C 180,E1 14238.362,E2 14238.362} C_VEL
LIN {X 0,Y 402.69,Z 513.685,A -85,B 0,C 180,E1 14235.777,E2 14235.777} C_VEL
LIN {X 0,Y 399.532,Z 508.91,A -85,B 0,C 180,E1 14233.902,E2 14233.902} C_VEL
LIN {X 0,Y 397.13,Z 505.283,A -85,B 0,C 180,E1 14232.284,E2 14232.284} C_VEL
LIN {X 0,Y 393.987,Z 500.614,A -85,B 0,C 180,E1 14229.79,E2 14229.79} C_VEL
LIN {X 0,Y 391.246,Z 496.487,A -85,B 0,C 180,E1 14226.973,E2 14226.973} C_VEL
LIN {X 0,Y 390.728,Z 495.704,A -85,B 0,C 180,E1 14226.318,E2 14226.318} C_VEL
LIN {X 0,Y 388.012,Z 490.465,A -85,B 0,C 180,E1 14218.671,E2 14218.671} C_VEL
LIN {X 0,Y 391.156,Z 496.248,A -85,B 0,C 180,E1 14210.732,E2 14210.732} C_VEL
LIN {X 0,Y 394.104,Z 500.734,A -85,B 0,C 180,E1 14207.695,E2 14207.695} C_VEL
LIN {X 0,Y 398.294,Z 507.008,A -85,B 0,C 180,E1 14204.493,E2 14204.493} C_VEL
LIN {X 0,Y 401.9,Z 512.442,A -85,B 0,C 180,E1 14202.256,E2 14202.256} C_VEL
LIN {X 0,Y 406.635,Z 519.608,A -85,B 0,C 180,E1 14199.751,E2 14199.751} C_VEL
LIN {X 0,Y 412.649,Z 529.458,A -85,B 0,C 180,E1 14197,E2 14197} C_VEL
LIN {X 0,Y 419.569,Z 541.223,A -85,B 0,C 180,E1 14194.261,E2 14194.261} C_VEL
LIN {X 0,Y 420.876,Z 543.854,A -85,B 0,C 180,E1 14193.769,E2 14193.769} C_VEL
LIN {X 0,Y 404.626,Z 746.959,A -85,B 0,C 180,E1 14190.458,E2 14190.458} C_VEL
LIN {X 0,Y 401.028,Z 773.491,A -85,B 0,C 180,E1 14189.868,E2 14189.868} C_VEL
LIN {X 0,Y 397.2,Z 794.082,A -85,B 0,C 180,E1 14189.255,E2 14189.255} C_VEL
LIN {X 0,Y 391.709,Z 817.882,A -85,B 0,C 180,E1 14188.354,E2 14188.354} C_VEL
LIN {X 0,Y 385.55,Z 839.656,A -85,B 0,C 180,E1 14187.305,E2 14187.305} C_VEL
LIN {X 0,Y 378.278,Z 862.046,A -85,B 0,C 180,E1 14185.987,E2 14185.987} C_VEL
LIN {X 0,Y 370.377,Z 882.821,A -85,B 0,C 180,E1 14184.483,E2 14184.483} C_VEL
LIN {X 0,Y 361.905,Z 903.106,A -85,B 0,C 180,E1 14182.721,E2 14182.721} C_VEL
LIN {X 0,Y 352.831,Z 922.417,A -85,B 0,C 180,E1 14180.683,E2 14180.683} C_VEL
LIN {X 0,Y 344.041,Z 939.832,A -85,B 0,C 180,E1 14178.498,E2 14178.498} C_VEL
LIN {X 0,Y 334.478,Z 957.369,A -85,B 0,C 180,E1 14175.845,E2 14175.845} C_VEL
LIN {X 0,Y 325.941,Z 972.191,A -85,B 0,C 180,E1 14173.165,E2 14173.165} C_VEL
LIN {X 0,Y 316.347,Z 988.176,A -85,B 0,C 180,E1 14169.678,E2 14169.678} C_VEL
LIN {X 0,Y 308.595,Z 1000.694,A -85,B 0,C 180,E1 14166.366,E2 14166.366} C_VEL
LIN {X 0,Y 300.833,Z 1013.275,A -85,B 0,C 180,E1 14162.352,E2 14162.352} C_VEL
LIN {X 0,Y 294.611,Z 1023.418,A -85,B 0,C 180,E1 14158.369,E2 14158.369} C_VEL
LIN {X 0,Y 289.198,Z 1032.87,A -85,B 0,C 180,E1 14153.861,E2 14153.861} C_VEL
LIN {X 0,Y 285.183,Z 1040.428,A -85,B 0,C 180,E1 14149.243,E2 14149.243} C_VEL
LIN {X 0,Y 282.487,Z 1046.527,A -85,B 0,C 180,E1 14144.555,E2 14144.555} C_VEL
LIN {X 0,Y 280.863,Z 1051.135,A -85,B 0,C 180,E1 14139.632,E2 14139.632} C_VEL
LIN {X 0,Y 280.246,Z 1053.806,A -85,B 0,C 180,E1 14135.528,E2 14135.528} C_VEL
LIN {X 0,Y 280.034,Z 1055.508,A -85,B 0,C 180,E1 14131.215,E2 14131.215} C_VEL
LIN {X 0,Y 280.003,Z 1055.98,A -85,B 0,C 180,E1 14126.725,E2 14126.725} C_VEL
LIN {X 0,Y 280.119,Z 1055.275,A -85,B 0,C 180,E1 14122.617,E2 14122.617} C_VEL
LIN {X 0,Y 280.485,Z 1053.606,A -85,B 0,C 180,E1 14118.62,E2 14118.62} C_VEL
LIN {X 0,Y 281.592,Z 1050.422,A -85,B 0,C 180,E1 14113.921,E2 14113.921} C_VEL
LIN {X 0,Y 283.879,Z 1045.321,A -85,B 0,C 180,E1 14108.945,E2 14108.945} C_VEL
LIN {X 0,Y 287.209,Z 1039.23,A -85,B 0,C 180,E1 14104.425,E2 14104.425} C_VEL
LIN {X 0,Y 292.452,Z 1030.6,A -85,B 0,C 180,E1 14099.496,E2 14099.496} C_VEL
LIN {X 0,Y 298.182,Z 1021.813,A -85,B 0,C 180,E1 14095.479,E2 14095.479} C_VEL
LIN {X 0,Y 306.424,Z 1009.502,A -85,B 0,C 180,E1 14090.952,E2 14090.952} C_VEL
LIN {X 0,Y 314.05,Z 998.143,A -85,B 0,C 180,E1 14087.548,E2 14087.548} C_VEL
LIN {X 0,Y 324.098,Z 982.835,A -85,B 0,C 180,E1 14083.786,E2 14083.786} C_VEL
LIN {X 0,Y 332.708,Z 969.207,A -85,B 0,C 180,E1 14081.033,E2 14081.033} C_VEL
LIN {X 0,Y 343.144,Z 951.871,A -85,B 0,C 180,E1 14078.117,E2 14078.117} C_VEL
LIN {X 0,Y 352.231,Z 935.616,A -85,B 0,C 180,E1 14075.859,E2 14075.859} C_VEL
LIN {X 0,Y 361.829,Z 917.319,A -85,B 0,C 180,E1 14073.717,E2 14073.717} C_VEL
LIN {X 0,Y 370.857,Z 898.112,A -85,B 0,C 180,E1 14071.865,E2 14071.865} C_VEL
LIN {X 0,Y 378.885,Z 879.443,A -85,B 0,C 180,E1 14070.349,E2 14070.349} C_VEL
LIN {X 0,Y 387.606,Z 856.479,A -85,B 0,C 180,E1 14068.82,E2 14068.82} C_VEL
LIN {X 0,Y 394.201,Z 836.465,A -85,B 0,C 180,E1 14067.719,E2 14067.719} C_VEL
LIN {X 0,Y 401.217,Z 811.37,A -85,B 0,C 180,E1 14066.613,E2 14066.613} C_VEL
LIN {X 0,Y 406.128,Z 789.851,A -85,B 0,C 180,E1 14065.87,E2 14065.87} C_VEL
LIN {X 0,Y 410.704,Z 764.047,A -85,B 0,C 180,E1 14065.19,E2 14065.19} C_VEL
LIN {X 0,Y 413.436,Z 741.716,A -85,B 0,C 180,E1 14064.755,E2 14064.755} C_VEL
LIN {X 0,Y 415.705,Z 715.097,A -85,B 0,C 180,E1 14064.319,E2 14064.319} C_VEL
LIN {X 0,Y 415.899,Z 707.54,A -85,B 0,C 180,E1 14064.074,E2 14064.074} C_VEL
LIN {X 0,Y 414.928,Z 687.872,A -85,B 0,C 180,E1 14062.973,E2 14062.973} C_VEL
LIN {X 0,Y 415.159,Z 681.375,A -85,B 0,C 180,E1 14062.772,E2 14062.772} C_VEL
LIN {X 0,Y 425.901,Z 554.4,A -85,B 0,C 180,E1 14060.763,E2 14060.763} C_VEL
LIN {X 0,Y 419.442,Z 543.145,A -85,B 0,C 180,E1 14057.838,E2 14057.838} C_VEL
LIN {X 0,Y 414.203,Z 534.559,A -85,B 0,C 180,E1 14055.041,E2 14055.041} C_VEL
LIN {X 0,Y 410.956,Z 529.462,A -85,B 0,C 180,E1 14053.007,E2 14053.007} C_VEL
LIN {X 0,Y 408.862,Z 526.106,A -85,B 0,C 180,E1 14051.497,E2 14051.497} C_VEL
LIN {X 0,Y 406.319,Z 522.059,A -85,B 0,C 180,E1 14049.347,E2 14049.347} C_VEL
LIN {X 0,Y 403.45,Z 517.419,A -85,B 0,C 180,E1 14046.118,E2 14046.118} C_VEL
LIN {X 0,Y 401.055,Z 512.724,A -85,B 0,C 180,E1 14039.143,E2 14039.143} C_VEL
LIN {X 0,Y 403.802,Z 517.98,A -85,B 0,C 180,E1 14031.743,E2 14031.743} C_VEL
LIN {X 0,Y 406.377,Z 522.134,A -85,B 0,C 180,E1 14028.935,E2 14028.935} C_VEL
LIN {X 0,Y 410.252,Z 528.245,A -85,B 0,C 180,E1 14025.821,E2 14025.821} C_VEL
LIN {X 0,Y 413.501,Z 533.436,A -85,B 0,C 180,E1 14023.71,E2 14023.71} C_VEL
LIN {X 0,Y 416.125,Z 537.897,A -85,B 0,C 180,E1 14022.196,E2 14022.196} C_VEL
LIN {X 0,Y 421.95,Z 549.263,A -85,B 0,C 180,E1 14019.215,E2 14019.215} C_VEL
LIN {X 0,Y 425.774,Z 557.6,A -85,B 0,C 180,E1 14017.471,E2 14017.471} C_VEL
LIN {X 0,Y 408.854,Z 756.627,A -85,B 0,C 180,E1 14014.291,E2 14014.291} C_VEL
LIN {X 0,Y 404.961,Z 783.408,A -85,B 0,C 180,E1 14013.74,E2 14013.74} C_VEL
LIN {X 0,Y 400.596,Z 804.942,A -85,B 0,C 180,E1 14013.167,E2 14013.167} C_VEL
LIN {X 0,Y 394.541,Z 828.877,A -85,B 0,C 180,E1 14012.343,E2 14012.343} C_VEL
LIN {X 0,Y 388.207,Z 849.575,A -85,B 0,C 180,E1 14011.438,E2 14011.438} C_VEL
LIN {X 0,Y 380.573,Z 871.453,A -85,B 0,C 180,E1 14010.265,E2 14010.265} C_VEL
LIN {X 0,Y 371.72,Z 893.243,A -85,B 0,C 180,E1 14008.803,E2 14008.803} C_VEL
LIN {X 0,Y 362.466,Z 913.79,A -85,B 0,C 180,E1 14007.139,E2 14007.139} C_VEL
LIN {X 0,Y 352.59,Z 933.381,A -85,B 0,C 180,E1 14005.183,E2 14005.183} C_VEL
LIN {X 0,Y 342.856,Z 951.283,A -85,B 0,C 180,E1 14003.042,E2 14003.042} C_VEL
LIN {X 0,Y 332.195,Z 969.387,A -85,B 0,C 180,E1 14000.403,E2 14000.403} C_VEL
LIN {X 0,Y 322.814,Z 984.464,A -85,B 0,C 180,E1 13997.755,E2 13997.755} C_VEL
LIN {X 0,Y 312.22,Z 1000.737,A -85,B 0,C 180,E1 13994.279,E2 13994.279} C_VEL
LIN {X 0,Y 303.63,Z 1013.532,A -85,B 0,C 180,E1 13990.945,E2 13990.945} C_VEL
LIN {X 0,Y 294.606,Z 1026.928,A -85,B 0,C 180,E1 13986.68,E2 13986.68} C_VEL
LIN {X 0,Y 288.02,Z 1036.849,A -85,B 0,C 180,E1 13982.791,E2 13982.791} C_VEL
LIN {X 0,Y 281.941,Z 1046.596,A -85,B 0,C 180,E1 13978.143,E2 13978.143} C_VEL
LIN {X 0,Y 277.43,Z 1054.442,A -85,B 0,C 180,E1 13973.357,E2 13973.357} C_VEL
LIN {X 0,Y 274.416,Z 1060.8,A -85,B 0,C 180,E1 13968.482,E2 13968.482} C_VEL
LIN {X 0,Y 272.672,Z 1065.618,A -85,B 0,C 180,E1 13963.357,E2 13963.357} C_VEL
LIN {X 0,Y 272.073,Z 1068.433,A -85,B 0,C 180,E1 13959.092,E2 13959.092} C_VEL
LIN {X 0,Y 271.968,Z 1070.223,A -85,B 0,C 180,E1 13954.639,E2 13954.639} C_VEL
LIN {X 0,Y 272.005,Z 1070.724,A -85,B 0,C 180,E1 13950.211,E2 13950.211} C_VEL
LIN {X 0,Y 271.975,Z 1070.003,A -85,B 0,C 180,E1 13945.995,E2 13945.995} C_VEL
LIN {X 0,Y 272.005,Z 1068.413,A -85,B 0,C 180,E1 13942.183,E2 13942.183} C_VEL
LIN {X 0,Y 272.412,Z 1065.575,A -85,B 0,C 180,E1 13937.923,E2 13937.923} C_VEL
LIN {X 0,Y 273.802,Z 1060.673,A -85,B 0,C 180,E1 13932.794,E2 13932.794} C_VEL
LIN {X 0,Y 276.24,Z 1054.546,A -85,B 0,C 180,E1 13928.11,E2 13928.11} C_VEL
LIN {X 0,Y 280.198,Z 1046.645,A -85,B 0,C 180,E1 13923.28,E2 13923.28} C_VEL
LIN {X 0,Y 285.703,Z 1036.797,A -85,B 0,C 180,E1 13918.57,E2 13918.57} C_VEL
LIN {X 0,Y 292.115,Z 1026.242,A -85,B 0,C 180,E1 13914.416,E2 13914.416} C_VEL
LIN {X 0,Y 300.214,Z 1013.16,A -85,B 0,C 180,E1 13910.247,E2 13910.247} C_VEL
LIN {X 0,Y 308.335,Z 1000.179,A -85,B 0,C 180,E1 13906.824,E2 13906.824} C_VEL
LIN {X 0,Y 317.943,Z 984.437,A -85,B 0,C 180,E1 13903.409,E2 13903.409} C_VEL
LIN {X 0,Y 326.365,Z 970.121,A -85,B 0,C 180,E1 13900.823,E2 13900.823} C_VEL
LIN {X 0,Y 336.576,Z 951.917,A -85,B 0,C 180,E1 13898.071,E2 13898.071} C_VEL
LIN {X 0,Y 345.635,Z 934.474,A -85,B 0,C 180,E1 13895.903,E2 13895.903} C_VEL
LIN {X 0,Y 355.169,Z 914.815,A -85,B 0,C 180,E1 13893.85,E2 13893.85} C_VEL
LIN {X 0,Y 364.176,Z 894.039,A -85,B 0,C 180,E1 13892.091,E2 13892.091} C_VEL
LIN {X 0,Y 372.39,Z 873.151,A -85,B 0,C 180,E1 13890.62,E2 13890.62} C_VEL
LIN {X 0,Y 379.814,Z 851.354,A -85,B 0,C 180,E1 13889.38,E2 13889.38} C_VEL
LIN {X 0,Y 385.604,Z 831.934,A -85,B 0,C 180,E1 13888.473,E2 13888.473} C_VEL
LIN {X 0,Y 391.89,Z 806.962,A -85,B 0,C 180,E1 13887.547,E2 13887.547} C_VEL
LIN {X 0,Y 396.291,Z 784.838,A -85,B 0,C 180,E1 13886.924,E2 13886.924} C_VEL
LIN {X 0,Y 399.998,Z 759.664,A -85,B 0,C 180,E1 13886.373,E2 13886.373} C_VEL
LIN {X 0,Y 405.251,Z 696.996,A -85,B 0,C 180,E1 13885.326,E2 13885.326} C_VEL
LIN {X 0,Y 417.039,Z 551.019,A -85,B 0,C 180,E1 13882.954,E2 13882.954} C_VEL
LIN {X 0,Y 410.551,Z 537.832,A -85,B 0,C 180,E1 13880.233,E2 13880.233} C_VEL
LIN {X 0,Y 405.662,Z 528.531,A -85,B 0,C 180,E1 13877.908,E2 13877.908} C_VEL
LIN {X 0,Y 400.833,Z 520.865,A -85,B 0,C 180,E1 13875.333,E2 13875.333} C_VEL
LIN {X 0,Y 397.667,Z 515.967,A -85,B 0,C 180,E1 13873.375,E2 13873.375} C_VEL
LIN {X 0,Y 395.548,Z 512.727,A -85,B 0,C 180,E1 13871.889,E2 13871.889} C_VEL
LIN {X 0,Y 392.677,Z 508.329,A -85,B 0,C 180,E1 13869.527,E2 13869.527} C_VEL
LIN {X 0,Y 390.029,Z 504.17,A -85,B 0,C 180,E1 13866.699,E2 13866.699} C_VEL
LIN {X 0,Y 387.041,Z 498.372,A -85,B 0,C 180,E1 13858.808,E2 13858.808} C_VEL
LIN {X 0,Y 390,Z 504.074,A -85,B 0,C 180,E1 13850.928,E2 13850.928} C_VEL
LIN {X 0,Y 392.797,Z 508.455,A -85,B 0,C 180,E1 13847.952,E2 13847.952} C_VEL
LIN {X 0,Y 396.79,Z 514.56,A -85,B 0,C 180,E1 13844.807,E2 13844.807} C_VEL
LIN {X 0,Y 400.43,Z 520.187,A -85,B 0,C 180,E1 13842.489,E2 13842.489} C_VEL
LIN {X 0,Y 404.947,Z 527.232,A -85,B 0,C 180,E1 13840.04,E2 13840.04} C_VEL
LIN {X 0,Y 410.799,Z 537.02,A -85,B 0,C 180,E1 13837.299,E2 13837.299} C_VEL
LIN {X 0,Y 417.195,Z 548.17,A -85,B 0,C 180,E1 13834.698,E2 13834.698} C_VEL
LIN {X 0,Y 400.877,Z 747.136,A -85,B 0,C 180,E1 13831.465,E2 13831.465} C_VEL
LIN {X 0,Y 397.205,Z 773.682,A -85,B 0,C 180,E1 13830.878,E2 13830.878} C_VEL
LIN {X 0,Y 393.285,Z 794.342,A -85,B 0,C 180,E1 13830.268,E2 13830.268} C_VEL
LIN {X 0,Y 387.58,Z 818.48,A -85,B 0,C 180,E1 13829.358,E2 13829.358} C_VEL
LIN {X 0,Y 381.633,Z 839.09,A -85,B 0,C 180,E1 13828.376,E2 13828.376} C_VEL
LIN {X 0,Y 374.467,Z 860.832,A -85,B 0,C 180,E1 13827.115,E2 13827.115} C_VEL
LIN {X 0,Y 366.098,Z 882.48,A -85,B 0,C 180,E1 13825.571,E2 13825.571} C_VEL
LIN {X 0,Y 357.715,Z 902.093,A -85,B 0,C 180,E1 13823.883,E2 13823.883} C_VEL
LIN {X 0,Y 348.074,Z 922.218,A -85,B 0,C 180,E1 13821.782,E2 13821.782} C_VEL
LIN {X 0,Y 339.196,Z 939.334,A -85,B 0,C 180,E1 13819.642,E2 13819.642} C_VEL
LIN {X 0,Y 328.874,Z 957.728,A -85,B 0,C 180,E1 13816.86,E2 13816.86} C_VEL
LIN {X 0,Y 320.057,Z 972.539,A -85,B 0,C 180,E1 13814.161,E2 13814.161} C_VEL
LIN {X 0,Y 310.124,Z 988.502,A -85,B 0,C 180,E1 13810.638,E2 13810.638} C_VEL
LIN {X 0,Y 302.469,Z 1000.386,A -85,B 0,C 180,E1 13807.464,E2 13807.464} C_VEL
LIN {X 0,Y 294.314,Z 1013.068,A -85,B 0,C 180,E1 13803.392,E2 13803.392} C_VEL
LIN {X 0,Y 287.583,Z 1023.513,A -85,B 0,C 180,E1 13799.226,E2 13799.226} C_VEL
LIN {X 0,Y 281.991,Z 1032.783,A -85,B 0,C 180,E1 13794.734,E2 13794.734} C_VEL
LIN {X 0,Y 277.652,Z 1040.456,A -85,B 0,C 180,E1 13789.961,E2 13789.961} C_VEL
LIN {X 0,Y 274.859,Z 1046.286,A -85,B 0,C 180,E1 13785.4,E2 13785.4} C_VEL
LIN {X 0,Y 272.983,Z 1051.219,A -85,B 0,C 180,E1 13780.126,E2 13780.126} C_VEL
LIN {X 0,Y 272.285,Z 1053.927,A -85,B 0,C 180,E1 13775.902,E2 13775.902} C_VEL
LIN {X 0,Y 272.046,Z 1055.594,A -85,B 0,C 180,E1 13771.685,E2 13771.685} C_VEL
LIN {X 0,Y 272.003,Z 1056.234,A -85,B 0,C 180,E1 13767.05,E2 13767.05} C_VEL
LIN {X 0,Y 272.124,Z 1055.545,A -85,B 0,C 180,E1 13762.611,E2 13762.611} C_VEL
LIN {X 0,Y 272.518,Z 1053.875,A -85,B 0,C 180,E1 13758.422,E2 13758.422} C_VEL
LIN {X 0,Y 273.601,Z 1050.926,A -85,B 0,C 180,E1 13753.874,E2 13753.874} C_VEL
LIN {X 0,Y 276.088,Z 1045.75,A -85,B 0,C 180,E1 13748.544,E2 13748.544} C_VEL
LIN {X 0,Y 279.397,Z 1039.998,A -85,B 0,C 180,E1 13744.112,E2 13744.112} C_VEL
LIN {X 0,Y 285.094,Z 1031.139,A -85,B 0,C 180,E1 13738.845,E2 13738.845} C_VEL
LIN {X 0,Y 291.056,Z 1022.416,A -85,B 0,C 180,E1 13734.75,E2 13734.75} C_VEL
LIN {X 0,Y 299.612,Z 1010.235,A -85,B 0,C 180,E1 13730.152,E2 13730.152} C_VEL
LIN {X 0,Y 307.537,Z 998.894,A -85,B 0,C 180,E1 13726.684,E2 13726.684} C_VEL
LIN {X 0,Y 317.43,Z 984.468,A -85,B 0,C 180,E1 13723.047,E2 13723.047} C_VEL
LIN {X 0,Y 326.803,Z 970.137,A -85,B 0,C 180,E1 13720.102,E2 13720.102} C_VEL
LIN {X 0,Y 336.958,Z 953.954,A -85,B 0,C 180,E1 13717.32,E2 13717.32} C_VEL
LIN {X 0,Y 346.802,Z 936.885,A -85,B 0,C 180,E1 13714.918,E2 13714.918} C_VEL
LIN {X 0,Y 356.043,Z 919.785,A -85,B 0,C 180,E1 13712.892,E2 13712.892} C_VEL
LIN {X 0,Y 365.943,Z 899.567,A -85,B 0,C 180,E1 13710.91,E2 13710.91} C_VEL
LIN {X 0,Y 374.138,Z 881.037,A -85,B 0,C 180,E1 13709.397,E2 13709.397} C_VEL
LIN {X 0,Y 383.305,Z 857.667,A -85,B 0,C 180,E1 13707.833,E2 13707.833} C_VEL
LIN {X 0,Y 390.133,Z 837.471,A -85,B 0,C 180,E1 13706.724,E2 13706.724} C_VEL
LIN {X 0,Y 397.109,Z 813.363,A -85,B 0,C 180,E1 13705.655,E2 13705.655} C_VEL
LIN {X 0,Y 402.273,Z 791.391,A -85,B 0,C 180,E1 13704.894,E2 13704.894} C_VEL
LIN {X 0,Y 406.787,Z 767.391,A -85,B 0,C 180,E1 13704.249,E2 13704.249} C_VEL
LIN {X 0,Y 409.842,Z 743.575,A -85,B 0,C 180,E1 13703.778,E2 13703.778} C_VEL
LIN {X 0,Y 415.159,Z 681.375,A -85,B 0,C 180,E1 13702.772,E2 13702.772} C_VEL
LIN {X 0,Y 415.386,Z 673.823,A -85,B 0,C 180,E1 13702.524,E2 13702.524} C_VEL
LIN {X 0,Y 414.627,Z 654.162,A -85,B 0,C 180,E1 13701.417,E2 13701.417} C_VEL
LIN {X 0,Y 414.9,Z 647.667,A -85,B 0,C 180,E1 13701.218,E2 13701.218} C_VEL
LIN {X 0,Y 422.541,Z 559.274,A -85,B 0,C 180,E1 13699.815,E2 13699.815} C_VEL
LIN {X 0,Y 416.843,Z 549.22,A -85,B 0,C 180,E1 13697.088,E2 13697.088} C_VEL
LIN {X 0,Y 412.069,Z 541.213,A -85,B 0,C 180,E1 13694.402,E2 13694.402} C_VEL
LIN {X 0,Y 407.973,Z 534.388,A -85,B 0,C 180,E1 13691.594,E2 13691.594} C_VEL
LIN {X 0,Y 405.035,Z 529.771,A -85,B 0,C 180,E1 13689.091,E2 13689.091} C_VEL
LIN {X 0,Y 402.367,Z 525.305,A -85,B 0,C 180,E1 13685.991,E2 13685.991} C_VEL
LIN {X 0,Y 400.08,Z 520.669,A -85,B 0,C 180,E1 13679.141,E2 13679.141} C_VEL
LIN {X 0,Y 402.66,Z 525.801,A -85,B 0,C 180,E1 13671.935,E2 13671.935} C_VEL
LIN {X 0,Y 405.249,Z 530.019,A -85,B 0,C 180,E1 13669.048,E2 13669.048} C_VEL
LIN {X 0,Y 408.874,Z 535.96,A -85,B 0,C 180,E1 13666.062,E2 13666.062} C_VEL
LIN {X 0,Y 412.058,Z 541.171,A -85,B 0,C 180,E1 13663.941,E2 13663.941} C_VEL
LIN {X 0,Y 414.568,Z 545.618,A -85,B 0,C 180,E1 13662.453,E2 13662.453} C_VEL
LIN {X 0,Y 419.938,Z 556.451,A -85,B 0,C 180,E1 13659.621,E2 13659.621} C_VEL
LIN {X 0,Y 422.458,Z 562.256,A -85,B 0,C 180,E1 13658.408,E2 13658.408} C_VEL
LIN {X 0,Y 405.55,Z 756.488,A -85,B 0,C 180,E1 13655.321,E2 13655.321} C_VEL
LIN {X 0,Y 401.596,Z 783.183,A -85,B 0,C 180,E1 13654.776,E2 13654.776} C_VEL
LIN {X 0,Y 397.168,Z 804.654,A -85,B 0,C 180,E1 13654.213,E2 13654.213} C_VEL
LIN {X 0,Y 390.88,Z 829.007,A -85,B 0,C 180,E1 13653.385,E2 13653.385} C_VEL
LIN {X 0,Y 384.797,Z 848.536,A -85,B 0,C 180,E1 13652.546,E2 13652.546} C_VEL
LIN {X 0,Y 376.997,Z 870.507,A -85,B 0,C 180,E1 13651.389,E2 13651.389} C_VEL
LIN {X 0,Y 367.944,Z 892.434,A -85,B 0,C 180,E1 13649.943,E2 13649.943} C_VEL
LIN {X 0,Y 359.151,Z 911.567,A -85,B 0,C 180,E1 13648.421,E2 13648.421} C_VEL
LIN {X 0,Y 348.624,Z 932.171,A -85,B 0,C 180,E1 13646.412,E2 13646.412} C_VEL
LIN {X 0,Y 339.031,Z 949.387,A -85,B 0,C 180,E1 13644.384,E2 13644.384} C_VEL
LIN {X 0,Y 327.607,Z 968.363,A -85,B 0,C 180,E1 13641.664,E2 13641.664} C_VEL
LIN {X 0,Y 317.878,Z 983.509,A -85,B 0,C 180,E1 13639.019,E2 13639.019} C_VEL
LIN {X 0,Y 306.832,Z 999.938,A -85,B 0,C 180,E1 13635.522,E2 13635.522} C_VEL
LIN {X 0,Y 297.875,Z 1012.757,A -85,B 0,C 180,E1 13632.171,E2 13632.171} C_VEL
LIN {X 0,Y 288.76,Z 1025.735,A -85,B 0,C 180,E1 13628.051,E2 13628.051} C_VEL
LIN {X 0,Y 281.408,Z 1036.225,A -85,B 0,C 180,E1 13623.907,E2 13623.907} C_VEL
LIN {X 0,Y 274.916,Z 1046.06,A -85,B 0,C 180,E1 13619.168,E2 13619.168} C_VEL
LIN {X 0,Y 270.052,Z 1053.953,A -85,B 0,C 180,E1 13614.267,E2 13614.267} C_VEL
LIN {X 0,Y 266.872,Z 1060.095,A -85,B 0,C 180,E1 13609.479,E2 13609.479} C_VEL
LIN {X 0,Y 264.805,Z 1065.257,A -85,B 0,C 180,E1 13603.985,E2 13603.985} C_VEL
LIN {X 0,Y 264.108,Z 1068.114,A -85,B 0,C 180,E1 13599.589,E2 13599.589} C_VEL
LIN {X 0,Y 263.971,Z 1069.877,A -85,B 0,C 180,E1 13595.216,E2 13595.216} C_VEL
LIN {X 0,Y 264.002,Z 1070.551,A -85,B 0,C 180,E1 13590.651,E2 13590.651} C_VEL
LIN {X 0,Y 263.978,Z 1069.85,A -85,B 0,C 180,E1 13586.091,E2 13586.091} C_VEL
LIN {X 0,Y 264.016,Z 1068.183,A -85,B 0,C 180,E1 13581.945,E2 13581.945} C_VEL
LIN {X 0,Y 264.469,Z 1065.337,A -85,B 0,C 180,E1 13577.555,E2 13577.555} C_VEL
LIN {X 0,Y 265.983,Z 1060.421,A -85,B 0,C 180,E1 13572.272,E2 13572.272} C_VEL
LIN {X 0,Y 268.609,Z 1054.286,A -85,B 0,C 180,E1 13567.455,E2 13567.455} C_VEL
LIN {X 0,Y 272.852,Z 1046.342,A -85,B 0,C 180,E1 13562.478,E2 13562.478} C_VEL
LIN {X 0,Y 278.653,Z 1036.514,A -85,B 0,C 180,E1 13557.68,E2 13557.68} C_VEL
LIN {X 0,Y 285.398,Z 1025.951,A -85,B 0,C 180,E1 13553.445,E2 13553.445} C_VEL
LIN {X 0,Y 293.875,Z 1012.853,A -85,B 0,C 180,E1 13549.212,E2 13549.212} C_VEL
LIN {X 0,Y 302.339,Z 999.862,A -85,B 0,C 180,E1 13545.748,E2 13545.748} C_VEL
LIN {X 0,Y 312.68,Z 983.49,A -85,B 0,C 180,E1 13542.186,E2 13542.186} C_VEL
LIN {X 0,Y 321.585,Z 968.835,A -85,B 0,C 180,E1 13539.548,E2 13539.548} C_VEL
LIN {X 0,Y 332.759,Z 949.297,A -85,B 0,C 180,E1 13536.65,E2 13536.65} C_VEL
LIN {X 0,Y 341.818,Z 932.27,A -85,B 0,C 180,E1 13534.576,E2 13534.576} C_VEL
LIN {X 0,Y 352.329,Z 910.696,A -85,B 0,C 180,E1 13532.404,E2 13532.404} C_VEL
LIN {X 0,Y 360.6,Z 891.945,A -85,B 0,C 180,E1 13530.863,E2 13530.863} C_VEL
LIN {X 0,Y 369.484,Z 869.422,A -85,B 0,C 180,E1 13529.329,E2 13529.329} C_VEL
LIN {X 0,Y 376.626,Z 848.549,A -85,B 0,C 180,E1 13528.187,E2 13528.187} C_VEL
LIN {X 0,Y 383.323,Z 826.187,A -85,B 0,C 180,E1 13527.191,E2 13527.191} C_VEL
LIN {X 0,Y 388.947,Z 802.957,A -85,B 0,C 180,E1 13526.391,E2 13526.391} C_VEL
LIN {X 0,Y 393.386,Z 780.337,A -85,B 0,C 180,E1 13525.783,E2 13525.783} C_VEL
LIN {X 0,Y 396.831,Z 754.948,A -85,B 0,C 180,E1 13525.262,E2 13525.262} C_VEL
LIN {X 0,Y 413.463,Z 555.447,A -85,B 0,C 180,E1 13522.015,E2 13522.015} C_VEL
LIN {X 0,Y 407.879,Z 543.86,A -85,B 0,C 180,E1 13519.55,E2 13519.55} C_VEL
LIN {X 0,Y 403.629,Z 535.552,A -85,B 0,C 180,E1 13517.443,E2 13517.443} C_VEL
LIN {X 0,Y 399.117,Z 528.224,A -85,B 0,C 180,E1 13514.954,E2 13514.954} C_VEL
LIN {X 0,Y 395.939,Z 523.174,A -85,B 0,C 180,E1 13512.914,E2 13512.914} C_VEL
LIN {X 0,Y 394.08,Z 520.288,A -85,B 0,C 180,E1 13511.563,E2 13511.563} C_VEL
LIN {X 0,Y 391.375,Z 516.041,A -85,B 0,C 180,E1 13509.262,E2 13509.262} C_VEL
LIN {X 0,Y 388.773,Z 511.721,A -85,B 0,C 180,E1 13506.349,E2 13506.349} C_VEL
LIN {X 0,Y 386.056,Z 506.398,A -85,B 0,C 180,E1 13498.664,E2 13498.664} C_VEL
LIN {X 0,Y 388.849,Z 511.898,A -85,B 0,C 180,E1 13491.125,E2 13491.125} C_VEL
LIN {X 0,Y 391.663,Z 516.343,A -85,B 0,C 180,E1 13488.066,E2 13488.066} C_VEL
LIN {X 0,Y 395.503,Z 522.476,A -85,B 0,C 180,E1 13484.974,E2 13484.974} C_VEL
LIN {X 0,Y 399.083,Z 528.109,A -85,B 0,C 180,E1 13482.653,E2 13482.653} C_VEL
LIN {X 0,Y 403.868,Z 535.881,A -85,B 0,C 180,E1 13480.022,E2 13480.022} C_VEL
LIN {X 0,Y 409.546,Z 545.579,A -85,B 0,C 180,E1 13477.344,E2 13477.344} C_VEL
LIN {X 0,Y 413.587,Z 552.965,A -85,B 0,C 180,E1 13475.636,E2 13475.636} C_VEL
LIN {X 0,Y 397.244,Z 747.418,A -85,B 0,C 180,E1 13472.488,E2 13472.488} C_VEL
LIN {X 0,Y 393.508,Z 773.872,A -85,B 0,C 180,E1 13471.908,E2 13471.908} C_VEL
LIN {X 0,Y 389.503,Z 794.561,A -85,B 0,C 180,E1 13471.303,E2 13471.303} C_VEL
LIN {X 0,Y 383.572,Z 819.078,A -85,B 0,C 180,E1 13470.385,E2 13470.385} C_VEL
LIN {X 0,Y 377.502,Z 839.643,A -85,B 0,C 180,E1 13469.41,E2 13469.41} C_VEL
LIN {X 0,Y 370.179,Z 861.348,A -85,B 0,C 180,E1 13468.157,E2 13468.157} C_VEL
LIN {X 0,Y 361.567,Z 883.06,A -85,B 0,C 180,E1 13466.611,E2 13466.611} C_VEL
LIN {X 0,Y 352.648,Z 903.392,A -85,B 0,C 180,E1 13464.859,E2 13464.859} C_VEL
LIN {X 0,Y 342.827,Z 923.22,A -85,B 0,C 180,E1 13462.772,E2 13462.772} C_VEL
LIN {X 0,Y 333.395,Z 940.87,A -85,B 0,C 180,E1 13460.545,E2 13460.545} C_VEL
LIN {X 0,Y 322.96,Z 958.778,A -85,B 0,C 180,E1 13457.791,E2 13457.791} C_VEL
LIN {X 0,Y 313.764,Z 973.718,A -85,B 0,C 180,E1 13455.029,E2 13455.029} C_VEL
LIN {X 0,Y 303.526,Z 989.517,A -85,B 0,C 180,E1 13451.463,E2 13451.463} C_VEL
LIN {X 0,Y 295.212,Z 1001.951,A -85,B 0,C 180,E1 13448.056,E2 13448.056} C_VEL
LIN {X 0,Y 286.477,Z 1014.88,A -85,B 0,C 180,E1 13443.708,E2 13443.708} C_VEL
LIN {X 0,Y 280.076,Z 1024.445,A -85,B 0,C 180,E1 13439.751,E2 13439.751} C_VEL
LIN {X 0,Y 273.93,Z 1034.106,A -85,B 0,C 180,E1 13434.82,E2 13434.82} C_VEL
LIN {X 0,Y 269.738,Z 1041.252,A -85,B 0,C 180,E1 13430.166,E2 13430.166} C_VEL
LIN {X 0,Y 266.65,Z 1047.491,A -85,B 0,C 180,E1 13424.995,E2 13424.995} C_VEL
LIN {X 0,Y 264.949,Z 1051.769,A -85,B 0,C 180,E1 13419.997,E2 13419.997} C_VEL
LIN {X 0,Y 264.265,Z 1054.38,A -85,B 0,C 180,E1 13415.646,E2 13415.646} C_VEL
LIN {X 0,Y 264.029,Z 1056.114,A -85,B 0,C 180,E1 13410.651,E2 13410.651} C_VEL
LIN {X 0,Y 264.015,Z 1056.357,A -85,B 0,C 180,E1 13406.091,E2 13406.091} C_VEL
LIN {X 0,Y 264.155,Z 1055.619,A -85,B 0,C 180,E1 13401.949,E2 13401.949} C_VEL
LIN {X 0,Y 264.623,Z 1053.931,A -85,B 0,C 180,E1 13397.784,E2 13397.784} C_VEL
LIN {X 0,Y 266.023,Z 1050.613,A -85,B 0,C 180,E1 13392.689,E2 13392.689} C_VEL
LIN {X 0,Y 268.588,Z 1045.68,A -85,B 0,C 180,E1 13387.684,E2 13387.684} C_VEL
LIN {X 0,Y 272.399,Z 1039.575,A -85,B 0,C 180,E1 13382.924,E2 13382.924} C_VEL
LIN {X 0,Y 278.174,Z 1031.101,A -85,B 0,C 180,E1 13377.86,E2 13377.86} C_VEL
LIN {X 0,Y 284.319,Z 1022.565,A -85,B 0,C 180,E1 13373.785,E2 13373.785} C_VEL
LIN {X 0,Y 293.288,Z 1010.366,A -85,B 0,C 180,E1 13369.113,E2 13369.113} C_VEL
LIN {X 0,Y 301.557,Z 999.016,A -85,B 0,C 180,E1 13365.603,E2 13365.603} C_VEL
LIN {X 0,Y 311.843,Z 984.569,A -85,B 0,C 180,E1 13361.937,E2 13361.937} C_VEL
LIN {X 0,Y 321.55,Z 970.226,A -85,B 0,C 180,E1 13358.977,E2 13358.977} C_VEL
LIN {X 0,Y 332.159,Z 953.804,A -85,B 0,C 180,E1 13356.158,E2 13356.158} C_VEL
LIN {X 0,Y 342.234,Z 936.819,A -85,B 0,C 180,E1 13353.777,E2 13353.777} C_VEL
LIN {X 0,Y 352.025,Z 919.162,A -85,B 0,C 180,E1 13351.7,E2 13351.7} C_VEL
LIN {X 0,Y 361.813,Z 899.568,A -85,B 0,C 180,E1 13349.801,E2 13349.801} C_VEL
LIN {X 0,Y 369.855,Z 881.819,A -85,B 0,C 180,E1 13348.36,E2 13348.36} C_VEL
LIN {X 0,Y 378.855,Z 859.592,A -85,B 0,C 180,E1 13346.866,E2 13346.866} C_VEL
LIN {X 0,Y 385.95,Z 839.194,A -85,B 0,C 180,E1 13345.743,E2 13345.743} C_VEL
LIN {X 0,Y 392.93,Z 816.1,A -85,B 0,C 180,E1 13344.707,E2 13344.707} C_VEL
LIN {X 0,Y 398.61,Z 792.605,A -85,B 0,C 180,E1 13343.89,E2 13343.89} C_VEL
LIN {X 0,Y 403.197,Z 769.107,A -85,B 0,C 180,E1 13343.255,E2 13343.255} C_VEL
LIN {X 0,Y 406.468,Z 744.491,A -85,B 0,C 180,E1 13342.766,E2 13342.766} C_VEL
LIN {X 0,Y 414.9,Z 647.667,A -85,B 0,C 180,E1 13341.218,E2 13341.218} C_VEL
LIN {X 0,Y 415.176,Z 640.115,A -85,B 0,C 180,E1 13340.97,E2 13340.97} C_VEL
LIN {X 0,Y 414.623,Z 620.462,A -85,B 0,C 180,E1 13339.857,E2 13339.857} C_VEL
LIN {X 0,Y 414.936,Z 613.966,A -85,B 0,C 180,E1 13339.659,E2 13339.659} C_VEL
LIN {X 0,Y 419.36,Z 564.343,A -85,B 0,C 180,E1 13338.885,E2 13338.885} C_VEL
LIN {X 0,Y 413.72,Z 554.136,A -85,B 0,C 180,E1 13335.993,E2 13335.993} C_VEL
LIN {X 0,Y 408.97,Z 546.064,A -85,B 0,C 180,E1 13333.071,E2 13333.071} C_VEL
LIN {X 0,Y 405.997,Z 541.23,A -85,B 0,C 180,E1 13330.86,E2 13330.86} C_VEL
LIN {X 0,Y 403.759,Z 537.481,A -85,B 0,C 180,E1 13328.832,E2 13328.832} C_VEL
LIN {X 0,Y 401.18,Z 533.109,A -85,B 0,C 180,E1 13325.722,E2 13325.722} C_VEL
LIN {X 0,Y 399.103,Z 528.618,A -85,B 0,C 180,E1 13319.139,E2 13319.139} C_VEL
LIN {X 0,Y 401.522,Z 533.618,A -85,B 0,C 180,E1 13312.128,E2 13312.128} C_VEL
LIN {X 0,Y 404.548,Z 538.8,A -85,B 0,C 180,E1 13308.74,E2 13308.74} C_VEL
LIN {X 0,Y 407.596,Z 543.839,A -85,B 0,C 180,E1 13306.234,E2 13306.234} C_VEL
LIN {X 0,Y 410.841,Z 549.26,A -85,B 0,C 180,E1 13304.037,E2 13304.037} C_VEL
LIN {X 0,Y 413.597,Z 554.533,A -85,B 0,C 180,E1 13302.374,E2 13302.374} C_VEL
LIN {X 0,Y 418.407,Z 564.676,A -85,B 0,C 180,E1 13299.799,E2 13299.799} C_VEL
LIN {X 0,Y 419.27,Z 566.769,A -85,B 0,C 180,E1 13299.363,E2 13299.363} C_VEL
LIN {X 0,Y 402.379,Z 756.349,A -85,B 0,C 180,E1 13296.367,E2 13296.367} C_VEL
LIN {X 0,Y 398.355,Z 783.014,A -85,B 0,C 180,E1 13295.829,E2 13295.829} C_VEL
LIN {X 0,Y 393.875,Z 804.37,A -85,B 0,C 180,E1 13295.277,E2 13295.277} C_VEL
LIN {X 0,Y 387.35,Z 829.141,A -85,B 0,C 180,E1 13294.447,E2 13294.447} C_VEL
LIN {X 0,Y 380.773,Z 849.756,A -85,B 0,C 180,E1 13293.566,E2 13293.566} C_VEL
LIN {X 0,Y 372.452,Z 872.443,A -85,B 0,C 180,E1 13292.365,E2 13292.365} C_VEL
LIN {X 0,Y 363.591,Z 893.249,A -85,B 0,C 180,E1 13290.987,E2 13290.987} C_VEL
LIN {X 0,Y 353.746,Z 914.085,A -85,B 0,C 180,E1 13289.32,E2 13289.32} C_VEL
LIN {X 0,Y 343.195,Z 933.886,A -85,B 0,C 180,E1 13287.351,E2 13287.351} C_VEL
LIN {X 0,Y 332.307,Z 952.812,A -85,B 0,C 180,E1 13285.078,E2 13285.078} C_VEL
LIN {X 0,Y 321.361,Z 970.13,A -85,B 0,C 180,E1 13282.506,E2 13282.506} C_VEL
LIN {X 0,Y 310.847,Z 985.952,A -85,B 0,C 180,E1 13279.672,E2 13279.672} C_VEL
LIN {X 0,Y 300.095,Z 1001.191,A -85,B 0,C 180,E1 13276.305,E2 13276.305} C_VEL
LIN {X 0,Y 290.873,Z 1013.903,A -85,B 0,C 180,E1 13272.893,E2 13272.893} C_VEL
LIN {X 0,Y 281.093,Z 1027.145,A -85,B 0,C 180,E1 13268.499,E2 13268.499} C_VEL
LIN {X 0,Y 273.756,Z 1037.209,A -85,B 0,C 180,E1 13264.364,E2 13264.364} C_VEL
LIN {X 0,Y 266.454,Z 1047.686,A -85,B 0,C 180,E1 13258.952,E2 13258.952} C_VEL
LIN {X 0,Y 262.003,Z 1054.7,A -85,B 0,C 180,E1 13254.341,E2 13254.341} C_VEL
LIN {X 0,Y 258.361,Z 1061.504,A -85,B 0,C 180,E1 13248.525,E2 13248.525} C_VEL
LIN {X 0,Y 256.739,Z 1065.554,A -85,B 0,C 180,E1 13243.743,E2 13243.743} C_VEL
LIN {X 0,Y 256.063,Z 1068.423,A -85,B 0,C 180,E1 13238.91,E2 13238.91} C_VEL
LIN {X 0,Y 255.972,Z 1069.995,A -85,B 0,C 180,E1 13234.032,E2 13234.032} C_VEL
LIN {X 0,Y 256.011,Z 1070.223,A -85,B 0,C 180,E1 13229.552,E2 13229.552} C_VEL
LIN {X 0,Y 255.978,Z 1069.488,A -85,B 0,C 180,E1 13225.519,E2 13225.519} C_VEL
LIN {X 0,Y 256.043,Z 1067.836,A -85,B 0,C 180,E1 13221.466,E2 13221.466} C_VEL
LIN {X 0,Y 256.577,Z 1064.934,A -85,B 0,C 180,E1 13216.937,E2 13216.937} C_VEL
LIN {X 0,Y 258.386,Z 1059.646,A -85,B 0,C 180,E1 13211.265,E2 13211.265} C_VEL
LIN {X 0,Y 261.178,Z 1053.714,A -85,B 0,C 180,E1 13206.537,E2 13206.537} C_VEL
LIN {X 0,Y 265.753,Z 1045.722,A -85,B 0,C 180,E1 13201.456,E2 13201.456} C_VEL
LIN {X 0,Y 271.893,Z 1035.899,A -85,B 0,C 180,E1 13196.595,E2 13196.595} C_VEL
LIN {X 0,Y 279.514,Z 1024.592,A -85,B 0,C 180,E1 13192.027,E2 13192.027} C_VEL
LIN {X 0,Y 288.077,Z 1011.898,A -85,B 0,C 180,E1 13187.942,E2 13187.942} C_VEL
LIN {X 0,Y 297.444,Z 998.121,A -85,B 0,C 180,E1 13184.273,E2 13184.273} C_VEL
LIN {X 0,Y 307.334,Z 982.906,A -85,B 0,C 180,E1 13180.993,E2 13180.993} C_VEL
LIN {X 0,Y 317.323,Z 966.988,A -85,B 0,C 180,E1 13178.141,E2 13178.141} C_VEL
LIN {X 0,Y 328.221,Z 948.363,A -85,B 0,C 180,E1 13175.422,E2 13175.422} C_VEL
LIN {X 0,Y 337.928,Z 930.566,A -85,B 0,C 180,E1 13173.278,E2 13173.278} C_VEL
LIN {X 0,Y 348.354,Z 909.534,A -85,B 0,C 180,E1 13171.201,E2 13171.201} C_VEL
LIN {X 0,Y 356.783,Z 890.808,A -85,B 0,C 180,E1 13169.683,E2 13169.683} C_VEL
LIN {X 0,Y 366.174,Z 867.228,A -85,B 0,C 180,E1 13168.116,E2 13168.116} C_VEL
LIN {X 0,Y 373.231,Z 846.885,A -85,B 0,C 180,E1 13167.03,E2 13167.03} C_VEL
LIN {X 0,Y 380.238,Z 823.446,A -85,B 0,C 180,E1 13166.024,E2 13166.024} C_VEL
LIN {X 0,Y 385.56,Z 801.659,A -85,B 0,C 180,E1 13165.297,E2 13165.297} C_VEL
LIN {X 0,Y 390.306,Z 777.572,A -85,B 0,C 180,E1 13164.669,E2 13164.669} C_VEL
LIN {X 0,Y 393.539,Z 752.897,A -85,B 0,C 180,E1 13164.18,E2 13164.18} C_VEL
LIN {X 0,Y 410.004,Z 559.968,A -85,B 0,C 180,E1 13161.064,E2 13161.064} C_VEL
LIN {X 0,Y 405.405,Z 550.158,A -85,B 0,C 180,E1 13158.925,E2 13158.925} C_VEL
LIN {X 0,Y 401.623,Z 542.572,A -85,B 0,C 180,E1 13156.972,E2 13156.972} C_VEL
LIN {X 0,Y 397.306,Z 535.4,A -85,B 0,C 180,E1 13154.502,E2 13154.502} C_VEL
LIN {X 0,Y 393.39,Z 528.806,A -85,B 0,C 180,E1 13151.807,E2 13151.807} C_VEL
LIN {X 0,Y 390.082,Z 523.752,A -85,B 0,C 180,E1 13148.996,E2 13148.996} C_VEL
LIN {X 0,Y 387.344,Z 519.272,A -85,B 0,C 180,E1 13145.778,E2 13145.778} C_VEL
LIN {X 0,Y 385.078,Z 514.364,A -85,B 0,C 180,E1 13138.661,E2 13138.661} C_VEL
LIN {X 0,Y 387.752,Z 519.847,A -85,B 0,C 180,E1 13131.249,E2 13131.249} C_VEL
LIN {X 0,Y 390.984,Z 525.13,A -85,B 0,C 180,E1 13127.745,E2 13127.745} C_VEL
LIN {X 0,Y 394.105,Z 530.18,A -85,B 0,C 180,E1 13125.227,E2 13125.227} C_VEL
LIN {X 0,Y 397.509,Z 535.663,A -85,B 0,C 180,E1 13122.96,E2 13122.96} C_VEL
LIN {X 0,Y 402.393,Z 543.816,A -85,B 0,C 180,E1 13120.211,E2 13120.211} C_VEL
LIN {X 0,Y 407.755,Z 553.293,A -85,B 0,C 180,E1 13117.623,E2 13117.623} C_VEL
LIN {X 0,Y 410.091,Z 557.754,A -85,B 0,C 180,E1 13116.589,E2 13116.589} C_VEL
LIN {X 0,Y 393.75,Z 747.589,A -85,B 0,C 180,E1 13113.531,E2 13113.531} C_VEL
LIN {X 0,Y 389.94,Z 774.061,A -85,B 0,C 180,E1 13112.957,E2 13112.957} C_VEL
LIN {X 0,Y 385.842,Z 794.82,A -85,B 0,C 180,E1 13112.357,E2 13112.357} C_VEL
LIN {X 0,Y 380.057,Z 818.404,A -85,B 0,C 180,E1 13111.488,E2 13111.488} C_VEL
LIN {X 0,Y 373.496,Z 840.196,A -85,B 0,C 180,E1 13110.466,E2 13110.466} C_VEL
LIN {X 0,Y 365.661,Z 862.774,A -85,B 0,C 180,E1 13109.162,E2 13109.162} C_VEL
LIN {X 0,Y 357.137,Z 883.691,A -85,B 0,C 180,E1 13107.673,E2 13107.673} C_VEL
LIN {X 0,Y 347.807,Z 904.404,A -85,B 0,C 180,E1 13105.889,E2 13105.889} C_VEL
LIN {X 0,Y 338.006,Z 923.619,A -85,B 0,C 180,E1 13103.861,E2 13103.861} C_VEL
LIN {X 0,Y 328.041,Z 941.749,A -85,B 0,C 180,E1 13101.568,E2 13101.568} C_VEL
LIN {X 0,Y 317.428,Z 959.357,A -85,B 0,C 180,E1 13098.837,E2 13098.837} C_VEL
LIN {X 0,Y 308.072,Z 974.064,A -85,B 0,C 180,E1 13096.098,E2 13096.098} C_VEL
LIN {X 0,Y 297.471,Z 989.842,A -85,B 0,C 180,E1 13092.502,E2 13092.502} C_VEL
LIN {X 0,Y 288.838,Z 1002.266,A -85,B 0,C 180,E1 13089.053,E2 13089.053} C_VEL
LIN {X 0,Y 279.726,Z 1015.178,A -85,B 0,C 180,E1 13084.635,E2 13084.635} C_VEL
LIN {X 0,Y 273.027,Z 1024.734,A -85,B 0,C 180,E1 13080.601,E2 13080.601} C_VEL
LIN {X 0,Y 266.562,Z 1034.378,A -85,B 0,C 180,E1 13075.555,E2 13075.555} C_VEL
LIN {X 0,Y 262.128,Z 1041.515,A -85,B 0,C 180,E1 13070.778,E2 13070.778} C_VEL
LIN {X 0,Y 258.842,Z 1047.739,A -85,B 0,C 180,E1 13065.459,E2 13065.459} C_VEL
LIN {X 0,Y 257.024,Z 1052.009,A -85,B 0,C 180,E1 13060.309,E2 13060.309} C_VEL
LIN {X 0,Y 256.283,Z 1054.626,A -85,B 0,C 180,E1 13055.794,E2 13055.794} C_VEL
LIN {X 0,Y 256.033,Z 1056.331,A -85,B 0,C 180,E1 13050.671,E2 13050.671} C_VEL
LIN {X 0,Y 256.02,Z 1056.568,A -85,B 0,C 180,E1 13045.969,E2 13045.969} C_VEL
LIN {X 0,Y 256.16,Z 1055.889,A -85,B 0,C 180,E1 13041.922,E2 13041.922} C_VEL
LIN {X 0,Y 256.653,Z 1054.24,A -85,B 0,C 180,E1 13037.627,E2 13037.627} C_VEL
LIN {X 0,Y 258.148,Z 1050.947,A -85,B 0,C 180,E1 13032.334,E2 13032.334} C_VEL
LIN {X 0,Y 260.988,Z 1045.859,A -85,B 0,C 180,E1 13026.997,E2 13026.997} C_VEL
LIN {X 0,Y 265.062,Z 1039.748,A -85,B 0,C 180,E1 13022.111,E2 13022.111} C_VEL
LIN {X 0,Y 271.19,Z 1031.258,A -85,B 0,C 180,E1 13016.929,E2 13016.929} C_VEL
LIN {X 0,Y 277.802,Z 1022.544,A -85,B 0,C 180,E1 13012.698,E2 13012.698} C_VEL
LIN {X 0,Y 287.066,Z 1010.498,A -85,B 0,C 180,E1 13008.028,E2 13008.028} C_VEL
LIN {X 0,Y 295.691,Z 999.138,A -85,B 0,C 180,E1 13004.479,E2 13004.479} C_VEL
LIN {X 0,Y 306.633,Z 984.305,A -85,B 0,C 180,E1 13000.706,E2 13000.706} C_VEL
LIN {X 0,Y 316.473,Z 970.246,A -85,B 0,C 180,E1 12997.803,E2 12997.803} C_VEL
LIN {X 0,Y 327.547,Z 953.575,A -85,B 0,C 180,E1 12994.951,E2 12994.951} C_VEL
LIN {X 0,Y 337.882,Z 936.625,A -85,B 0,C 180,E1 12992.588,E2 12992.588} C_VEL
LIN {X 0,Y 348.112,Z 918.633,A -85,B 0,C 180,E1 12990.492,E2 12990.492} C_VEL
LIN {X 0,Y 358.177,Z 898.826,A -85,B 0,C 180,E1 12988.603,E2 12988.603} C_VEL
LIN {X 0,Y 366.425,Z 880.976,A -85,B 0,C 180,E1 12987.18,E2 12987.18} C_VEL
LIN {X 0,Y 376,Z 857.489,A -85,B 0,C 180,E1 12985.645,E2 12985.645} C_VEL
LIN {X 0,Y 382.742,Z 838.351,A -85,B 0,C 180,E1 12984.615,E2 12984.615} C_VEL
LIN {X 0,Y 389.928,Z 814.657,A -85,B 0,C 180,E1 12983.58,E2 12983.58} C_VEL
LIN {X 0,Y 395.432,Z 792.19,A -85,B 0,C 180,E1 12982.816,E2 12982.816} C_VEL
LIN {X 0,Y 400.132,Z 768.278,A -85,B 0,C 180,E1 12982.185,E2 12982.185} C_VEL
LIN {X 0,Y 403.365,Z 744.104,A -85,B 0,C 180,E1 12981.715,E2 12981.715} C_VEL
LIN {X 0,Y 414.936,Z 613.966,A -85,B 0,C 180,E1 12979.659,E2 12979.659} C_VEL
LIN {X 0,Y 415.264,Z 606.415,A -85,B 0,C 180,E1 12979.414,E2 12979.414} C_VEL
LIN {X 0,Y 414.927,Z 586.769,A -85,B 0,C 180,E1 12978.298,E2 12978.298} C_VEL
LIN {X 0,Y 415.264,Z 580.278,A -85,B 0,C 180,E1 12978.096,E2 12978.096} C_VEL
LIN {X 0,Y 416.222,Z 569.318,A -85,B 0,C 180,E1 12977.908,E2 12977.908} C_VEL
LIN {X 0,Y 411.401,Z 560.533,A -85,B 0,C 180,E1 12975.29,E2 12975.29} C_VEL
LIN {X 0,Y 407.273,Z 553.31,A -85,B 0,C 180,E1 12972.621,E2 12972.621} C_VEL
LIN {X 0,Y 404.584,Z 548.791,A -85,B 0,C 180,E1 12970.538,E2 12970.538} C_VEL
LIN {X 0,Y 402.491,Z 545.19,A -85,B 0,C 180,E1 12968.572,E2 12968.572} C_VEL
LIN {X 0,Y 400.103,Z 540.993,A -85,B 0,C 180,E1 12965.593,E2 12965.593} C_VEL
LIN {X 0,Y 398.126,Z 536.577,A -85,B 0,C 180,E1 12959.137,E2 12959.137} C_VEL
LIN {X 0,Y 400.435,Z 541.558,A -85,B 0,C 180,E1 12952.251,E2 12952.251} C_VEL
LIN {X 0,Y 403.262,Z 546.497,A -85,B 0,C 180,E1 12948.993,E2 12948.993} C_VEL
LIN {X 0,Y 406.231,Z 551.55,A -85,B 0,C 180,E1 12946.477,E2 12946.477} C_VEL
LIN {X 0,Y 409.879,Z 557.729,A -85,B 0,C 180,E1 12943.977,E2 12943.977} C_VEL
LIN {X 0,Y 414.596,Z 567.79,A -85,B 0,C 180,E1 12941.182,E2 12941.182} C_VEL
LIN {X 0,Y 416.169,Z 571.629,A -85,B 0,C 180,E1 12940.326,E2 12940.326} C_VEL
LIN {X 0,Y 399.355,Z 756.105,A -85,B 0,C 180,E1 12937.431,E2 12937.431} C_VEL
LIN {X 0,Y 395.26,Z 782.795,A -85,B 0,C 180,E1 12936.899,E2 12936.899} C_VEL
LIN {X 0,Y 390.72,Z 804.085,A -85,B 0,C 180,E1 12936.359,E2 12936.359} C_VEL
LIN {X 0,Y 384.16,Z 828.616,A -85,B 0,C 180,E1 12935.553,E2 12935.553} C_VEL
LIN {X 0,Y 377.647,Z 848.72,A -85,B 0,C 180,E1 12934.714,E2 12934.714} C_VEL
LIN {X 0,Y 369.54,Z 870.622,A -85,B 0,C 180,E1 12933.587,E2 12933.587} C_VEL
LIN {X 0,Y 360.105,Z 892.442,A -85,B 0,C 180,E1 12932.174,E2 12932.174} C_VEL
LIN {X 0,Y 350.198,Z 913.003,A -85,B 0,C 180,E1 12930.556,E2 12930.556} C_VEL
LIN {X 0,Y 339.56,Z 932.615,A -85,B 0,C 180,E1 12928.644,E2 12928.644} C_VEL
LIN {X 0,Y 329.348,Z 949.968,A -85,B 0,C 180,E1 12926.605,E2 12926.605} C_VEL
LIN {X 0,Y 317.272,Z 968.784,A -85,B 0,C 180,E1 12923.89,E2 12923.89} C_VEL
LIN {X 0,Y 306.74,Z 984.149,A -85,B 0,C 180,E1 12921.176,E2 12921.176} C_VEL
LIN {X 0,Y 294.977,Z 1000.361,A -85,B 0,C 180,E1 12917.643,E2 12917.643} C_VEL
LIN {X 0,Y 285.344,Z 1013.128,A -85,B 0,C 180,E1 12914.213,E2 12914.213} C_VEL
LIN {X 0,Y 275.066,Z 1026.474,A -85,B 0,C 180,E1 12909.775,E2 12909.775} C_VEL
LIN {X 0,Y 267.462,Z 1036.371,A -85,B 0,C 180,E1 12905.676,E2 12905.676} C_VEL
LIN {X 0,Y 260.037,Z 1046.435,A -85,B 0,C 180,E1 12900.502,E2 12900.502} C_VEL
LIN {X 0,Y 254.873,Z 1053.939,A -85,B 0,C 180,E1 12895.536,E2 12895.536} C_VEL
LIN {X 0,Y 251.062,Z 1060.483,A -85,B 0,C 180,E1 12890.03,E2 12890.03} C_VEL
LIN {X 0,Y 248.95,Z 1065.028,A -85,B 0,C 180,E1 12884.657,E2 12884.657} C_VEL
LIN {X 0,Y 248.14,Z 1067.83,A -85,B 0,C 180,E1 12879.978,E2 12879.978} C_VEL
LIN {X 0,Y 247.973,Z 1069.677,A -85,B 0,C 180,E1 12874.858,E2 12874.858} C_VEL
LIN {X 0,Y 248.021,Z 1070.052,A -85,B 0,C 180,E1 12870,E2 12870} C_VEL
LIN {X 0,Y 247.98,Z 1069.335,A -85,B 0,C 180,E1 12865.606,E2 12865.606} C_VEL
LIN {X 0,Y 248.046,Z 1067.723,A -85,B 0,C 180,E1 12861.422,E2 12861.422} C_VEL
LIN {X 0,Y 248.608,Z 1064.852,A -85,B 0,C 180,E1 12856.735,E2 12856.735} C_VEL
LIN {X 0,Y 250.517,Z 1059.654,A -85,B 0,C 180,E1 12850.896,E2 12850.896} C_VEL
LIN {X 0,Y 253.457,Z 1053.765,A -85,B 0,C 180,E1 12846.025,E2 12846.025} C_VEL
LIN {X 0,Y 258.258,Z 1045.839,A -85,B 0,C 180,E1 12840.802,E2 12840.802} C_VEL
LIN {X 0,Y 264.773,Z 1035.947,A -85,B 0,C 180,E1 12835.758,E2 12835.758} C_VEL
LIN {X 0,Y 272.617,Z 1024.843,A -85,B 0,C 180,E1 12831.157,E2 12831.157} C_VEL
LIN {X 0,Y 281.51,Z 1012.236,A -85,B 0,C 180,E1 12827.003,E2 12827.003} C_VEL
LIN {X 0,Y 290.686,Z 999.228,A -85,B 0,C 180,E1 12823.466,E2 12823.466} C_VEL
LIN {X 0,Y 301.404,Z 983.427,A -85,B 0,C 180,E1 12819.975,E2 12819.975} C_VEL
LIN {X 0,Y 310.715,Z 969.08,A -85,B 0,C 180,E1 12817.359,E2 12817.359} C_VEL
LIN {X 0,Y 322.23,Z 950.24,A -85,B 0,C 180,E1 12814.527,E2 12814.527} C_VEL
LIN {X 0,Y 332.107,Z 932.701,A -85,B 0,C 180,E1 12812.38,E2 12812.38} C_VEL
LIN {X 0,Y 342.777,Z 912.085,A -85,B 0,C 180,E1 12810.295,E2 12810.295} C_VEL
LIN {X 0,Y 351.733,Z 892.799,A -85,B 0,C 180,E1 12808.713,E2 12808.713} C_VEL
LIN {X 0,Y 360.925,Z 870.794,A -85,B 0,C 180,E1 12807.217,E2 12807.217} C_VEL
LIN {X 0,Y 368.85,Z 848.64,A -85,B 0,C 180,E1 12806.02,E2 12806.02} C_VEL
LIN {X 0,Y 375.632,Z 826.938,A -85,B 0,C 180,E1 12805.072,E2 12805.072} C_VEL
LIN {X 0,Y 381.657,Z 803.273,A -85,B 0,C 180,E1 12804.269,E2 12804.269} C_VEL
LIN {X 0,Y 386.132,Z 781.442,A -85,B 0,C 180,E1 12803.693,E2 12803.693} C_VEL
LIN {X 0,Y 389.923,Z 755.233,A -85,B 0,C 180,E1 12803.157,E2 12803.157} C_VEL
LIN {X 0,Y 406.625,Z 564.396,A -85,B 0,C 180,E1 12800.08,E2 12800.08} C_VEL
LIN {X 0,Y 401.997,Z 554.312,A -85,B 0,C 180,E1 12797.777,E2 12797.777} C_VEL
LIN {X 0,Y 398.968,Z 548.318,A -85,B 0,C 180,E1 12796.115,E2 12796.115} C_VEL
LIN {X 0,Y 393.945,Z 539.834,A -85,B 0,C 180,E1 12792.981,E2 12792.981} C_VEL
LIN {X 0,Y 391.273,Z 535.532,A -85,B 0,C 180,E1 12790.975,E2 12790.975} C_VEL
LIN {X 0,Y 388.797,Z 531.461,A -85,B 0,C 180,E1 12788.727,E2 12788.727} C_VEL
LIN {X 0,Y 386.261,Z 527.154,A -85,B 0,C 180,E1 12785.645,E2 12785.645} C_VEL
LIN {X 0,Y 384.1,Z 522.33,A -85,B 0,C 180,E1 12778.657,E2 12778.657} C_VEL
LIN {X 0,Y 386.609,Z 527.665,A -85,B 0,C 180,E1 12771.448,E2 12771.448} C_VEL
LIN {X 0,Y 389.681,Z 532.832,A -85,B 0,C 180,E1 12768.004,E2 12768.004} C_VEL
LIN {X 0,Y 392.724,Z 537.899,A -85,B 0,C 180,E1 12765.476,E2 12765.476} C_VEL
LIN {X 0,Y 396.174,Z 543.574,A -85,B 0,C 180,E1 12763.127,E2 12763.127} C_VEL
LIN {X 0,Y 401.256,Z 552.273,A -85,B 0,C 180,E1 12760.228,E2 12760.228} C_VEL
LIN {X 0,Y 406.716,Z 562.494,A -85,B 0,C 180,E1 12757.56,E2 12757.56} C_VEL
LIN {X 0,Y 390.378,Z 747.862,A -85,B 0,C 180,E1 12754.591,E2 12754.591} C_VEL
LIN {X 0,Y 386.482,Z 774.375,A -85,B 0,C 180,E1 12754.021,E2 12754.021} C_VEL
LIN {X 0,Y 382.309,Z 795.094,A -85,B 0,C 180,E1 12753.429,E2 12753.429} C_VEL
LIN {X 0,Y 376.312,Z 819,A -85,B 0,C 180,E1 12752.556,E2 12752.556} C_VEL
LIN {X 0,Y 369.952,Z 839.738,A -85,B 0,C 180,E1 12751.596,E2 12751.596} C_VEL
LIN {X 0,Y 362.342,Z 861.385,A -85,B 0,C 180,E1 12750.371,E2 12750.371} C_VEL
LIN {X 0,Y 353.391,Z 883.053,A -85,B 0,C 180,E1 12748.859,E2 12748.859} C_VEL
LIN {X 0,Y 344.717,Z 901.951,A -85,B 0,C 180,E1 12747.264,E2 12747.264} C_VEL
LIN {X 0,Y 334.301,Z 922.216,A -85,B 0,C 180,E1 12745.187,E2 12745.187} C_VEL
LIN {X 0,Y 324.931,Z 938.89,A -85,B 0,C 180,E1 12743.125,E2 12743.125} C_VEL
LIN {X 0,Y 313.331,Z 957.889,A -85,B 0,C 180,E1 12740.27,E2 12740.27} C_VEL
LIN {X 0,Y 303.522,Z 972.849,A -85,B 0,C 180,E1 12737.52,E2 12737.52} C_VEL
LIN {X 0,Y 292.511,Z 988.789,A -85,B 0,C 180,E1 12733.941,E2 12733.941} C_VEL
LIN {X 0,Y 283.453,Z 1001.333,A -85,B 0,C 180,E1 12730.471,E2 12730.471} C_VEL
